prgEM.stEL3446_IO_1.MDP5001_342_Input.MDP5001_342_I1_Channel_Overcurrent					:=	MDP5001_342_I1_Channel_Overcurrent_1;
prgEM.stEL3446_IO_1.MDP5001_342_Input.MDP5001_342_I1_Channel_Inaccurate_Current			:=	MDP5001_342_I1_Channel_Inaccurate_Current_1;
prgEM.stEL3446_IO_1.MDP5001_342_Input.MDP5001_342_I1_Channel_Current_Guard_Warning		:=	MDP5001_342_I1_Channel_Current_Guard_Warning_1;
prgEM.stEL3446_IO_1.MDP5001_342_Input.MDP5001_342_I1_Channel_Current_Guard_Error			:=	MDP5001_342_I1_Channel_Current_Guard_Error_1;
prgEM.stEL3446_IO_1.MDP5001_342_Input.MDP5001_342_I1_Channel_Apparent_Power_Guard_Warning	:=	MDP5001_342_I1_Channel_Apparent_Power_Guard_Warning_1;
prgEM.stEL3446_IO_1.MDP5001_342_Input.MDP5001_342_I1_Channel_Apparent_Power_Guard_Error	:=	MDP5001_342_I1_Channel_Apparent_Power_Guard_Error_1;
prgEM.stEL3446_IO_1.MDP5001_342_Input.MDP5001_342_I1_Channel_Active_Power_Guard_Warning	:=	MDP5001_342_I1_Channel_Active_Power_Guard_Warning_1;
prgEM.stEL3446_IO_1.MDP5001_342_Input.MDP5001_342_I1_Channel_Active_Power_Guard_Error		:=	MDP5001_342_I1_Channel_Active_Power_Guard_Error_1;
prgEM.stEL3446_IO_1.MDP5001_342_Input.MDP5001_342_I1_Channel_Reactive_Power_Guard_Warning	:=	MDP5001_342_I1_Channel_Reactive_Power_Guard_Warning_1;
prgEM.stEL3446_IO_1.MDP5001_342_Input.MDP5001_342_I1_Channel_Reactive_Power_Guard_Error	:=	MDP5001_342_I1_Channel_Reactive_Power_Guard_Error_1;
prgEM.stEL3446_IO_1.MDP5001_342_Input.MDP5001_342_I1_Channel_DPM_Inaccurate				:=	MDP5001_342_I1_Channel_DPM_Inaccurate_1;
prgEM.stEL3446_IO_1.MDP5001_342_Input.MDP5001_342_I1_Channel_DPM_Timeout					:=	MDP5001_342_I1_Channel_DPM_Timeout_1;
prgEM.stEL3446_IO_1.MDP5001_342_Input.MDP5001_342_I1_Channel_TxPDO_Toggle					:=	MDP5001_342_I1_Channel_TxPDO_Toggle_1;
prgEM.stEL3446_IO_1.MDP5001_342_Input.MDP5001_342_I1_Channel_Current						:=	MDP5001_342_I1_Channel_Current_1;
prgEM.stEL3446_IO_1.MDP5001_342_Input.MDP5001_342_I1_Channel_Active_Power					:=	MDP5001_342_I1_Channel_Active_Power_1;
prgEM.stEL3446_IO_1.MDP5001_342_Input.MDP5001_342_I1_Channel_Apparent_Power				:=	MDP5001_342_I1_Channel_Apparent_Power_1;
prgEM.stEL3446_IO_1.MDP5001_342_Input.MDP5001_342_I1_Channel_Reactive_Power_Fundamental	:=	MDP5001_342_I1_Channel_Reactive_Power_Fundamental_1;
prgEM.stEL3446_IO_1.MDP5001_342_Input.MDP5001_342_I1_Channel_Active_Energy				:=	MDP5001_342_I1_Channel_Active_Energy_1;
prgEM.stEL3446_IO_1.MDP5001_342_Input.MDP5001_342_I2_Channel_Overcurrent					:=	MDP5001_342_I2_Channel_Overcurrent_1;
prgEM.stEL3446_IO_1.MDP5001_342_Input.MDP5001_342_I2_Channel_Inaccurate_Current			:=	MDP5001_342_I2_Channel_Inaccurate_Current_1;
prgEM.stEL3446_IO_1.MDP5001_342_Input.MDP5001_342_I2_Channel_Current_Guard_Warning		:=	MDP5001_342_I2_Channel_Current_Guard_Warning_1;
prgEM.stEL3446_IO_1.MDP5001_342_Input.MDP5001_342_I2_Channel_Current_Guard_Error			:=	MDP5001_342_I2_Channel_Current_Guard_Error_1;
prgEM.stEL3446_IO_1.MDP5001_342_Input.MDP5001_342_I2_Channel_Apparent_Power_Guard_Warning	:=	MDP5001_342_I2_Channel_Apparent_Power_Guard_Warning_1;
prgEM.stEL3446_IO_1.MDP5001_342_Input.MDP5001_342_I2_Channel_Apparent_Power_Guard_Error	:=	MDP5001_342_I2_Channel_Apparent_Power_Guard_Error_1;
prgEM.stEL3446_IO_1.MDP5001_342_Input.MDP5001_342_I2_Channel_Active_Power_Guard_Warning	:=	MDP5001_342_I2_Channel_Active_Power_Guard_Warning_1;
prgEM.stEL3446_IO_1.MDP5001_342_Input.MDP5001_342_I2_Channel_Active_Power_Guard_Error		:=	MDP5001_342_I2_Channel_Active_Power_Guard_Error_1;
prgEM.stEL3446_IO_1.MDP5001_342_Input.MDP5001_342_I2_Channel_Reactive_Power_Guard_Warning	:=	MDP5001_342_I2_Channel_Reactive_Power_Guard_Warning_1;
prgEM.stEL3446_IO_1.MDP5001_342_Input.MDP5001_342_I2_Channel_Reactive_Power_Guard_Error	:=	MDP5001_342_I2_Channel_Reactive_Power_Guard_Error_1;
prgEM.stEL3446_IO_1.MDP5001_342_Input.MDP5001_342_I2_Channel_DPM_Inaccurate				:=	MDP5001_342_I2_Channel_DPM_Inaccurate_1;
prgEM.stEL3446_IO_1.MDP5001_342_Input.MDP5001_342_I2_Channel_DPM_Timeout					:=	MDP5001_342_I2_Channel_DPM_Timeout_1;
prgEM.stEL3446_IO_1.MDP5001_342_Input.MDP5001_342_I2_Channel_TxPDO_Toggle					:=	MDP5001_342_I2_Channel_TxPDO_Toggle_1;
prgEM.stEL3446_IO_1.MDP5001_342_Input.MDP5001_342_I2_Channel_Current						:=	MDP5001_342_I2_Channel_Current_1;
prgEM.stEL3446_IO_1.MDP5001_342_Input.MDP5001_342_I2_Channel_Active_Power					:=	MDP5001_342_I2_Channel_Active_Power_1;
prgEM.stEL3446_IO_1.MDP5001_342_Input.MDP5001_342_I2_Channel_Apparent_Power				:=	MDP5001_342_I2_Channel_Apparent_Power_1;
prgEM.stEL3446_IO_1.MDP5001_342_Input.MDP5001_342_I2_Channel_Reactive_Power_Fundamental	:=	MDP5001_342_I2_Channel_Reactive_Power_Fundamental_1;
prgEM.stEL3446_IO_1.MDP5001_342_Input.MDP5001_342_I2_Channel_Active_Energy				:=	MDP5001_342_I2_Channel_Active_Energy_1;
prgEM.stEL3446_IO_1.MDP5001_342_Input.MDP5001_342_I3_Channel_Overcurrent					:=	MDP5001_342_I3_Channel_Overcurrent_1;
prgEM.stEL3446_IO_1.MDP5001_342_Input.MDP5001_342_I3_Channel_Inaccurate_Current			:=	MDP5001_342_I3_Channel_Inaccurate_Current_1;
prgEM.stEL3446_IO_1.MDP5001_342_Input.MDP5001_342_I3_Channel_Current_Guard_Warning		:=	MDP5001_342_I3_Channel_Current_Guard_Warning_1;
prgEM.stEL3446_IO_1.MDP5001_342_Input.MDP5001_342_I3_Channel_Current_Guard_Error			:=	MDP5001_342_I3_Channel_Current_Guard_Error_1;
prgEM.stEL3446_IO_1.MDP5001_342_Input.MDP5001_342_I3_Channel_Apparent_Power_Guard_Warning	:=	MDP5001_342_I3_Channel_Apparent_Power_Guard_Warning_1;
prgEM.stEL3446_IO_1.MDP5001_342_Input.MDP5001_342_I3_Channel_Apparent_Power_Guard_Error	:=	MDP5001_342_I3_Channel_Apparent_Power_Guard_Error_1;
prgEM.stEL3446_IO_1.MDP5001_342_Input.MDP5001_342_I3_Channel_Active_Power_Guard_Warning	:=	MDP5001_342_I3_Channel_Active_Power_Guard_Warning_1;
prgEM.stEL3446_IO_1.MDP5001_342_Input.MDP5001_342_I3_Channel_Active_Power_Guard_Error		:=	MDP5001_342_I3_Channel_Active_Power_Guard_Error_1;
prgEM.stEL3446_IO_1.MDP5001_342_Input.MDP5001_342_I3_Channel_Reactive_Power_Guard_Warning	:=	MDP5001_342_I3_Channel_Reactive_Power_Guard_Warning_1;
prgEM.stEL3446_IO_1.MDP5001_342_Input.MDP5001_342_I3_Channel_Reactive_Power_Guard_Error	:=	MDP5001_342_I3_Channel_Reactive_Power_Guard_Error_1;
prgEM.stEL3446_IO_1.MDP5001_342_Input.MDP5001_342_I3_Channel_DPM_Inaccurate				:=	MDP5001_342_I3_Channel_DPM_Inaccurate_1;
prgEM.stEL3446_IO_1.MDP5001_342_Input.MDP5001_342_I3_Channel_DPM_Timeout					:=	MDP5001_342_I3_Channel_DPM_Timeout_1;
prgEM.stEL3446_IO_1.MDP5001_342_Input.MDP5001_342_I3_Channel_TxPDO_Toggle					:=	MDP5001_342_I3_Channel_TxPDO_Toggle_1;
prgEM.stEL3446_IO_1.MDP5001_342_Input.MDP5001_342_I3_Channel_Current						:=	MDP5001_342_I3_Channel_Current_1;
prgEM.stEL3446_IO_1.MDP5001_342_Input.MDP5001_342_I3_Channel_Active_Power					:=	MDP5001_342_I3_Channel_Active_Power_1;
prgEM.stEL3446_IO_1.MDP5001_342_Input.MDP5001_342_I3_Channel_Apparent_Power				:=	MDP5001_342_I3_Channel_Apparent_Power_1;
prgEM.stEL3446_IO_1.MDP5001_342_Input.MDP5001_342_I3_Channel_Reactive_Power_Fundamental	:=	MDP5001_342_I3_Channel_Reactive_Power_Fundamental_1;
prgEM.stEL3446_IO_1.MDP5001_342_Input.MDP5001_342_I3_Channel_Active_Energy				:=	MDP5001_342_I3_Channel_Active_Energy_1;
prgEM.stEL3446_IO_1.MDP5001_342_Input.MDP5001_342_I4_Channel_Overcurrent					:=	MDP5001_342_I4_Channel_Overcurrent_1;
prgEM.stEL3446_IO_1.MDP5001_342_Input.MDP5001_342_I4_Channel_Inaccurate_Current			:=	MDP5001_342_I4_Channel_Inaccurate_Current_1;
prgEM.stEL3446_IO_1.MDP5001_342_Input.MDP5001_342_I4_Channel_Current_Guard_Warning		:=	MDP5001_342_I4_Channel_Current_Guard_Warning_1;
prgEM.stEL3446_IO_1.MDP5001_342_Input.MDP5001_342_I4_Channel_Current_Guard_Error			:=	MDP5001_342_I4_Channel_Current_Guard_Error_1;
prgEM.stEL3446_IO_1.MDP5001_342_Input.MDP5001_342_I4_Channel_Apparent_Power_Guard_Warning	:=	MDP5001_342_I4_Channel_Apparent_Power_Guard_Warning_1;
prgEM.stEL3446_IO_1.MDP5001_342_Input.MDP5001_342_I4_Channel_Apparent_Power_Guard_Error	:=	MDP5001_342_I4_Channel_Apparent_Power_Guard_Error_1;
prgEM.stEL3446_IO_1.MDP5001_342_Input.MDP5001_342_I4_Channel_Active_Power_Guard_Warning	:=	MDP5001_342_I4_Channel_Active_Power_Guard_Warning_1;
prgEM.stEL3446_IO_1.MDP5001_342_Input.MDP5001_342_I4_Channel_Active_Power_Guard_Error		:=	MDP5001_342_I4_Channel_Active_Power_Guard_Error_1;
prgEM.stEL3446_IO_1.MDP5001_342_Input.MDP5001_342_I4_Channel_Reactive_Power_Guard_Warning	:=	MDP5001_342_I4_Channel_Reactive_Power_Guard_Warning_1;
prgEM.stEL3446_IO_1.MDP5001_342_Input.MDP5001_342_I4_Channel_Reactive_Power_Guard_Error	:=	MDP5001_342_I4_Channel_Reactive_Power_Guard_Error_1;
prgEM.stEL3446_IO_1.MDP5001_342_Input.MDP5001_342_I4_Channel_DPM_Inaccurate				:=	MDP5001_342_I4_Channel_DPM_Inaccurate_1;
prgEM.stEL3446_IO_1.MDP5001_342_Input.MDP5001_342_I4_Channel_DPM_Timeout					:=	MDP5001_342_I4_Channel_DPM_Timeout_1;
prgEM.stEL3446_IO_1.MDP5001_342_Input.MDP5001_342_I4_Channel_TxPDO_Toggle					:=	MDP5001_342_I4_Channel_TxPDO_Toggle_1;
prgEM.stEL3446_IO_1.MDP5001_342_Input.MDP5001_342_I4_Channel_Current						:=	MDP5001_342_I4_Channel_Current_1;
prgEM.stEL3446_IO_1.MDP5001_342_Input.MDP5001_342_I4_Channel_Active_Power					:=	MDP5001_342_I4_Channel_Active_Power_1;
prgEM.stEL3446_IO_1.MDP5001_342_Input.MDP5001_342_I4_Channel_Apparent_Power				:=	MDP5001_342_I4_Channel_Apparent_Power_1;
prgEM.stEL3446_IO_1.MDP5001_342_Input.MDP5001_342_I4_Channel_Reactive_Power_Fundamental	:=	MDP5001_342_I4_Channel_Reactive_Power_Fundamental_1;
prgEM.stEL3446_IO_1.MDP5001_342_Input.MDP5001_342_I4_Channel_Active_Energy				:=	MDP5001_342_I4_Channel_Active_Energy_1;
prgEM.stEL3446_IO_1.MDP5001_342_Input.MDP5001_342_I5_Channel_Overcurrent					:=	MDP5001_342_I5_Channel_Overcurrent_1;
prgEM.stEL3446_IO_1.MDP5001_342_Input.MDP5001_342_I5_Channel_Inaccurate_Current			:=	MDP5001_342_I5_Channel_Inaccurate_Current_1;
prgEM.stEL3446_IO_1.MDP5001_342_Input.MDP5001_342_I5_Channel_Current_Guard_Warning		:=	MDP5001_342_I5_Channel_Current_Guard_Warning_1;
prgEM.stEL3446_IO_1.MDP5001_342_Input.MDP5001_342_I5_Channel_Current_Guard_Error			:=	MDP5001_342_I5_Channel_Current_Guard_Error_1;
prgEM.stEL3446_IO_1.MDP5001_342_Input.MDP5001_342_I5_Channel_Apparent_Power_Guard_Warning	:=	MDP5001_342_I5_Channel_Apparent_Power_Guard_Warning_1;
prgEM.stEL3446_IO_1.MDP5001_342_Input.MDP5001_342_I5_Channel_Apparent_Power_Guard_Error	:=	MDP5001_342_I5_Channel_Apparent_Power_Guard_Error_1;
prgEM.stEL3446_IO_1.MDP5001_342_Input.MDP5001_342_I5_Channel_Active_Power_Guard_Warning	:=	MDP5001_342_I5_Channel_Active_Power_Guard_Warning_1;
prgEM.stEL3446_IO_1.MDP5001_342_Input.MDP5001_342_I5_Channel_Active_Power_Guard_Error		:=	MDP5001_342_I5_Channel_Active_Power_Guard_Error_1;
prgEM.stEL3446_IO_1.MDP5001_342_Input.MDP5001_342_I5_Channel_Reactive_Power_Guard_Warning	:=	MDP5001_342_I5_Channel_Reactive_Power_Guard_Warning_1;
prgEM.stEL3446_IO_1.MDP5001_342_Input.MDP5001_342_I5_Channel_Reactive_Power_Guard_Error	:=	MDP5001_342_I5_Channel_Reactive_Power_Guard_Error_1;
prgEM.stEL3446_IO_1.MDP5001_342_Input.MDP5001_342_I5_Channel_DPM_Inaccurate				:=	MDP5001_342_I5_Channel_DPM_Inaccurate_1;
prgEM.stEL3446_IO_1.MDP5001_342_Input.MDP5001_342_I5_Channel_DPM_Timeout					:=	MDP5001_342_I5_Channel_DPM_Timeout_1;
prgEM.stEL3446_IO_1.MDP5001_342_Input.MDP5001_342_I5_Channel_TxPDO_Toggle					:=	MDP5001_342_I5_Channel_TxPDO_Toggle_1;
prgEM.stEL3446_IO_1.MDP5001_342_Input.MDP5001_342_I5_Channel_Current						:=	MDP5001_342_I5_Channel_Current_1;
prgEM.stEL3446_IO_1.MDP5001_342_Input.MDP5001_342_I5_Channel_Active_Power					:=	MDP5001_342_I5_Channel_Active_Power_1;
prgEM.stEL3446_IO_1.MDP5001_342_Input.MDP5001_342_I5_Channel_Apparent_Power				:=	MDP5001_342_I5_Channel_Apparent_Power_1;
prgEM.stEL3446_IO_1.MDP5001_342_Input.MDP5001_342_I5_Channel_Reactive_Power_Fundamental	:=	MDP5001_342_I5_Channel_Reactive_Power_Fundamental_1;
prgEM.stEL3446_IO_1.MDP5001_342_Input.MDP5001_342_I5_Channel_Active_Energy				:=	MDP5001_342_I5_Channel_Active_Energy_1;
prgEM.stEL3446_IO_1.MDP5001_342_Input.MDP5001_342_I6_Channel_Overcurrent					:=	MDP5001_342_I6_Channel_Overcurrent_1;
prgEM.stEL3446_IO_1.MDP5001_342_Input.MDP5001_342_I6_Channel_Inaccurate_Current			:=	MDP5001_342_I6_Channel_Inaccurate_Current_1;
prgEM.stEL3446_IO_1.MDP5001_342_Input.MDP5001_342_I6_Channel_Current_Guard_Warning		:=	MDP5001_342_I6_Channel_Current_Guard_Warning_1;
prgEM.stEL3446_IO_1.MDP5001_342_Input.MDP5001_342_I6_Channel_Current_Guard_Error			:=	MDP5001_342_I6_Channel_Current_Guard_Error_1;
prgEM.stEL3446_IO_1.MDP5001_342_Input.MDP5001_342_I6_Channel_Apparent_Power_Guard_Warning	:=	MDP5001_342_I6_Channel_Apparent_Power_Guard_Warning_1;
prgEM.stEL3446_IO_1.MDP5001_342_Input.MDP5001_342_I6_Channel_Apparent_Power_Guard_Error	:=	MDP5001_342_I6_Channel_Apparent_Power_Guard_Error_1;
prgEM.stEL3446_IO_1.MDP5001_342_Input.MDP5001_342_I6_Channel_Active_Power_Guard_Warning	:=	MDP5001_342_I6_Channel_Active_Power_Guard_Warning_1;
prgEM.stEL3446_IO_1.MDP5001_342_Input.MDP5001_342_I6_Channel_Active_Power_Guard_Error		:=	MDP5001_342_I6_Channel_Active_Power_Guard_Error_1;
prgEM.stEL3446_IO_1.MDP5001_342_Input.MDP5001_342_I6_Channel_Reactive_Power_Guard_Warning	:=	MDP5001_342_I6_Channel_Reactive_Power_Guard_Warning_1;
prgEM.stEL3446_IO_1.MDP5001_342_Input.MDP5001_342_I6_Channel_Reactive_Power_Guard_Error	:=	MDP5001_342_I6_Channel_Reactive_Power_Guard_Error_1;
prgEM.stEL3446_IO_1.MDP5001_342_Input.MDP5001_342_I6_Channel_DPM_Inaccurate				:=	MDP5001_342_I6_Channel_DPM_Inaccurate_1;
prgEM.stEL3446_IO_1.MDP5001_342_Input.MDP5001_342_I6_Channel_DPM_Timeout					:=	MDP5001_342_I6_Channel_DPM_Timeout_1;
prgEM.stEL3446_IO_1.MDP5001_342_Input.MDP5001_342_I6_Channel_TxPDO_Toggle					:=	MDP5001_342_I6_Channel_TxPDO_Toggle_1;
prgEM.stEL3446_IO_1.MDP5001_342_Input.MDP5001_342_I6_Channel_Current						:=	MDP5001_342_I6_Channel_Current_1;
prgEM.stEL3446_IO_1.MDP5001_342_Input.MDP5001_342_I6_Channel_Active_Power					:=	MDP5001_342_I6_Channel_Active_Power_1;
prgEM.stEL3446_IO_1.MDP5001_342_Input.MDP5001_342_I6_Channel_Apparent_Power				:=	MDP5001_342_I6_Channel_Apparent_Power_1;
prgEM.stEL3446_IO_1.MDP5001_342_Input.MDP5001_342_I6_Channel_Reactive_Power_Fundamental	:=	MDP5001_342_I6_Channel_Reactive_Power_Fundamental_1;
prgEM.stEL3446_IO_1.MDP5001_342_Input.MDP5001_342_I6_Channel_Active_Energy				:=	MDP5001_342_I6_Channel_Active_Energy_1;
prgEM.stEL3446_IO_1.MDP5001_342_Input.MDP5001_342_DPM_Variant_Value_In_TxPDO_Toggle		:=	MDP5001_342_DPM_Variant_Value_In_TxPDO_Toggle_1;
prgEM.stEL3446_IO_1.MDP5001_342_Input.MDP5001_342_DPM_Variant_Value_In_Index_1_REAL		:=	MDP5001_342_DPM_Variant_Value_In_Index_1_REAL_1;
prgEM.stEL3446_IO_1.MDP5001_342_Input.MDP5001_342_DPM_Variant_Value_In_Value_1_REAL		:=	MDP5001_342_DPM_Variant_Value_In_Value_1_REAL_1;
prgEM.stEL3446_IO_1.MDP5001_342_Input.MDP5001_342_DPM_Variant_Value_In_Index_2_REAL		:=	MDP5001_342_DPM_Variant_Value_In_Index_2_REAL_1;
prgEM.stEL3446_IO_1.MDP5001_342_Input.MDP5001_342_DPM_Variant_Value_In_Value_2_REAL		:=	MDP5001_342_DPM_Variant_Value_In_Value_2_REAL_1;
prgEM.stEL3446_IO_1.MDP5001_342_Input.MDP5001_342_DPM_Variant_Value_In_Index_3_REAL		:=	MDP5001_342_DPM_Variant_Value_In_Index_3_REAL_1;
prgEM.stEL3446_IO_1.MDP5001_342_Input.MDP5001_342_DPM_Variant_Value_In_Value_3_REAL		:=	MDP5001_342_DPM_Variant_Value_In_Value_3_REAL_1;
prgEM.stEL3446_IO_1.MDP5001_342_Input.MDP5001_342_DPM_Variant_Value_In_Index_4_ULINT		:=	MDP5001_342_DPM_Variant_Value_In_Index_4_ULINT_1;
prgEM.stEL3446_IO_1.MDP5001_342_Input.MDP5001_342_DPM_Variant_Value_In_Value_4_ULINT		:=	MDP5001_342_DPM_Variant_Value_In_Value_4_ULINT_1;

MDP5001_342_DPM_Variant_Value_Out_Index_1_REAL_1	:= 		prgEM.stEL3446_IO_1.MDP5001_342_Output.MDP5001_342_DPM_Variant_Value_Out_Index_1_REAL	;
MDP5001_342_DPM_Variant_Value_Out_Index_2_REAL_1	:= 		prgEM.stEL3446_IO_1.MDP5001_342_Output.MDP5001_342_DPM_Variant_Value_Out_Index_2_REAL	;	
MDP5001_342_DPM_Variant_Value_Out_Index_3_REAL_1	:= 		prgEM.stEL3446_IO_1.MDP5001_342_Output.MDP5001_342_DPM_Variant_Value_Out_Index_3_REAL	;
MDP5001_342_DPM_Variant_Value_Out_Index_4_ULINT_1	:= 		prgEM.stEL3446_IO_1.MDP5001_342_Output.MDP5001_342_DPM_Variant_Value_Out_Index_4_ULINT	;
MDP5001_342_DPM_Data_Data_1_1						:= 		prgEM.stEL3446_IO_1.MDP5001_342_Output.MDP5001_342_DPM_Data_Data_1	;
MDP5001_342_DPM_Data_Data_2_1						:= 		prgEM.stEL3446_IO_1.MDP5001_342_Output.MDP5001_342_DPM_Data_Data_2	;
MDP5001_342_DPM_Data_Data_3_1						:= 		prgEM.stEL3446_IO_1.MDP5001_342_Output.MDP5001_342_DPM_Data_Data_3	;
MDP5001_342_DPM_Data_Data_4_1						:= 		prgEM.stEL3446_IO_1.MDP5001_342_Output.MDP5001_342_DPM_Data_Data_4	;
MDP5001_342_DPM_Data_Data_5_1						:= 		prgEM.stEL3446_IO_1.MDP5001_342_Output.MDP5001_342_DPM_Data_Data_5	;
MDP5001_342_DPM_Data_Data_6_1						:= 		prgEM.stEL3446_IO_1.MDP5001_342_Output.MDP5001_342_DPM_Data_Data_6	;
MDP5001_342_DPM_Data_Data_7_1						:= 		prgEM.stEL3446_IO_1.MDP5001_342_Output.MDP5001_342_DPM_Data_Data_7	;
MDP5001_342_DPM_Data_Data_8_1						:= 		prgEM.stEL3446_IO_1.MDP5001_342_Output.MDP5001_342_DPM_Data_Data_8	;
MDP5001_342_DPM_Data_Data_9_1						:= 		prgEM.stEL3446_IO_1.MDP5001_342_Output.MDP5001_342_DPM_Data_Data_9	;
MDP5001_342_DPM_Data_Data_10_1						:= 		prgEM.stEL3446_IO_1.MDP5001_342_Output.MDP5001_342_DPM_Data_Data_10	;
MDP5001_342_DPM_Data_Data_11_1						:= 		prgEM.stEL3446_IO_1.MDP5001_342_Output.MDP5001_342_DPM_Data_Data_11	;
MDP5001_342_DPM_Data_Data_12_1						:= 		prgEM.stEL3446_IO_1.MDP5001_342_Output.MDP5001_342_DPM_Data_Data_12	;
MDP5001_342_DPM_Data_Data_13_1						:= 		prgEM.stEL3446_IO_1.MDP5001_342_Output.MDP5001_342_DPM_Data_Data_13	;
MDP5001_342_DPM_Data_Data_14_1						:= 		prgEM.stEL3446_IO_1.MDP5001_342_Output.MDP5001_342_DPM_Data_Data_14	;
MDP5001_342_DPM_Data_Data_15_1						:= 		prgEM.stEL3446_IO_1.MDP5001_342_Output.MDP5001_342_DPM_Data_Data_15	;
MDP5001_342_DPM_Data_Data_16_1						:= 		prgEM.stEL3446_IO_1.MDP5001_342_Output.MDP5001_342_DPM_Data_Data_16	;
MDP5001_342_DPM_Data_Data_17_1						:= 		prgEM.stEL3446_IO_1.MDP5001_342_Output.MDP5001_342_DPM_Data_Data_17	;
MDP5001_342_DPM_Data_Data_18_1						:= 		prgEM.stEL3446_IO_1.MDP5001_342_Output.MDP5001_342_DPM_Data_Data_18	;
MDP5001_342_DPM_Data_Data_19_1						:= 		prgEM.stEL3446_IO_1.MDP5001_342_Output.MDP5001_342_DPM_Data_Data_19	;
MDP5001_342_DPM_Data_Data_20_1						:= 		prgEM.stEL3446_IO_1.MDP5001_342_Output.MDP5001_342_DPM_Data_Data_20	;




prgEM.stEL3446_IO_2.MDP5001_342_Input.MDP5001_342_I1_Channel_Overcurrent					:=	MDP5001_342_I1_Channel_Overcurrent_2;
prgEM.stEL3446_IO_2.MDP5001_342_Input.MDP5001_342_I1_Channel_Inaccurate_Current			:=	MDP5001_342_I1_Channel_Inaccurate_Current_2;
prgEM.stEL3446_IO_2.MDP5001_342_Input.MDP5001_342_I1_Channel_Current_Guard_Warning		:=	MDP5001_342_I1_Channel_Current_Guard_Warning_2;
prgEM.stEL3446_IO_2.MDP5001_342_Input.MDP5001_342_I1_Channel_Current_Guard_Error			:=	MDP5001_342_I1_Channel_Current_Guard_Error_2;
prgEM.stEL3446_IO_2.MDP5001_342_Input.MDP5001_342_I1_Channel_Apparent_Power_Guard_Warning	:=	MDP5001_342_I1_Channel_Apparent_Power_Guard_Warning_2;
prgEM.stEL3446_IO_2.MDP5001_342_Input.MDP5001_342_I1_Channel_Apparent_Power_Guard_Error	:=	MDP5001_342_I1_Channel_Apparent_Power_Guard_Error_2;
prgEM.stEL3446_IO_2.MDP5001_342_Input.MDP5001_342_I1_Channel_Active_Power_Guard_Warning	:=	MDP5001_342_I1_Channel_Active_Power_Guard_Warning_2;
prgEM.stEL3446_IO_2.MDP5001_342_Input.MDP5001_342_I1_Channel_Active_Power_Guard_Error		:=	MDP5001_342_I1_Channel_Active_Power_Guard_Error_2;
prgEM.stEL3446_IO_2.MDP5001_342_Input.MDP5001_342_I1_Channel_Reactive_Power_Guard_Warning	:=	MDP5001_342_I1_Channel_Reactive_Power_Guard_Warning_2;
prgEM.stEL3446_IO_2.MDP5001_342_Input.MDP5001_342_I1_Channel_Reactive_Power_Guard_Error	:=	MDP5001_342_I1_Channel_Reactive_Power_Guard_Error_2;
prgEM.stEL3446_IO_2.MDP5001_342_Input.MDP5001_342_I1_Channel_DPM_Inaccurate				:=	MDP5001_342_I1_Channel_DPM_Inaccurate_2;
prgEM.stEL3446_IO_2.MDP5001_342_Input.MDP5001_342_I1_Channel_DPM_Timeout					:=	MDP5001_342_I1_Channel_DPM_Timeout_2;
prgEM.stEL3446_IO_2.MDP5001_342_Input.MDP5001_342_I1_Channel_TxPDO_Toggle					:=	MDP5001_342_I1_Channel_TxPDO_Toggle_2;
prgEM.stEL3446_IO_2.MDP5001_342_Input.MDP5001_342_I1_Channel_Current						:=	MDP5001_342_I1_Channel_Current_2;
prgEM.stEL3446_IO_2.MDP5001_342_Input.MDP5001_342_I1_Channel_Active_Power					:=	MDP5001_342_I1_Channel_Active_Power_2;
prgEM.stEL3446_IO_2.MDP5001_342_Input.MDP5001_342_I1_Channel_Apparent_Power				:=	MDP5001_342_I1_Channel_Apparent_Power_2;
prgEM.stEL3446_IO_2.MDP5001_342_Input.MDP5001_342_I1_Channel_Reactive_Power_Fundamental	:=	MDP5001_342_I1_Channel_Reactive_Power_Fundamental_2;
prgEM.stEL3446_IO_2.MDP5001_342_Input.MDP5001_342_I1_Channel_Active_Energy				:=	MDP5001_342_I1_Channel_Active_Energy_2;
prgEM.stEL3446_IO_2.MDP5001_342_Input.MDP5001_342_I2_Channel_Overcurrent					:=	MDP5001_342_I2_Channel_Overcurrent_2;
prgEM.stEL3446_IO_2.MDP5001_342_Input.MDP5001_342_I2_Channel_Inaccurate_Current			:=	MDP5001_342_I2_Channel_Inaccurate_Current_2;
prgEM.stEL3446_IO_2.MDP5001_342_Input.MDP5001_342_I2_Channel_Current_Guard_Warning		:=	MDP5001_342_I2_Channel_Current_Guard_Warning_2;
prgEM.stEL3446_IO_2.MDP5001_342_Input.MDP5001_342_I2_Channel_Current_Guard_Error			:=	MDP5001_342_I2_Channel_Current_Guard_Error_2;
prgEM.stEL3446_IO_2.MDP5001_342_Input.MDP5001_342_I2_Channel_Apparent_Power_Guard_Warning	:=	MDP5001_342_I2_Channel_Apparent_Power_Guard_Warning_2;
prgEM.stEL3446_IO_2.MDP5001_342_Input.MDP5001_342_I2_Channel_Apparent_Power_Guard_Error	:=	MDP5001_342_I2_Channel_Apparent_Power_Guard_Error_2;
prgEM.stEL3446_IO_2.MDP5001_342_Input.MDP5001_342_I2_Channel_Active_Power_Guard_Warning	:=	MDP5001_342_I2_Channel_Active_Power_Guard_Warning_2;
prgEM.stEL3446_IO_2.MDP5001_342_Input.MDP5001_342_I2_Channel_Active_Power_Guard_Error		:=	MDP5001_342_I2_Channel_Active_Power_Guard_Error_2;
prgEM.stEL3446_IO_2.MDP5001_342_Input.MDP5001_342_I2_Channel_Reactive_Power_Guard_Warning	:=	MDP5001_342_I2_Channel_Reactive_Power_Guard_Warning_2;
prgEM.stEL3446_IO_2.MDP5001_342_Input.MDP5001_342_I2_Channel_Reactive_Power_Guard_Error	:=	MDP5001_342_I2_Channel_Reactive_Power_Guard_Error_2;
prgEM.stEL3446_IO_2.MDP5001_342_Input.MDP5001_342_I2_Channel_DPM_Inaccurate				:=	MDP5001_342_I2_Channel_DPM_Inaccurate_2;
prgEM.stEL3446_IO_2.MDP5001_342_Input.MDP5001_342_I2_Channel_DPM_Timeout					:=	MDP5001_342_I2_Channel_DPM_Timeout_2;
prgEM.stEL3446_IO_2.MDP5001_342_Input.MDP5001_342_I2_Channel_TxPDO_Toggle					:=	MDP5001_342_I2_Channel_TxPDO_Toggle_2;
prgEM.stEL3446_IO_2.MDP5001_342_Input.MDP5001_342_I2_Channel_Current						:=	MDP5001_342_I2_Channel_Current_2;
prgEM.stEL3446_IO_2.MDP5001_342_Input.MDP5001_342_I2_Channel_Active_Power					:=	MDP5001_342_I2_Channel_Active_Power_2;
prgEM.stEL3446_IO_2.MDP5001_342_Input.MDP5001_342_I2_Channel_Apparent_Power				:=	MDP5001_342_I2_Channel_Apparent_Power_2;
prgEM.stEL3446_IO_2.MDP5001_342_Input.MDP5001_342_I2_Channel_Reactive_Power_Fundamental	:=	MDP5001_342_I2_Channel_Reactive_Power_Fundamental_2;
prgEM.stEL3446_IO_2.MDP5001_342_Input.MDP5001_342_I2_Channel_Active_Energy				:=	MDP5001_342_I2_Channel_Active_Energy_2;
prgEM.stEL3446_IO_2.MDP5001_342_Input.MDP5001_342_I3_Channel_Overcurrent					:=	MDP5001_342_I3_Channel_Overcurrent_2;
prgEM.stEL3446_IO_2.MDP5001_342_Input.MDP5001_342_I3_Channel_Inaccurate_Current			:=	MDP5001_342_I3_Channel_Inaccurate_Current_2;
prgEM.stEL3446_IO_2.MDP5001_342_Input.MDP5001_342_I3_Channel_Current_Guard_Warning		:=	MDP5001_342_I3_Channel_Current_Guard_Warning_2;
prgEM.stEL3446_IO_2.MDP5001_342_Input.MDP5001_342_I3_Channel_Current_Guard_Error			:=	MDP5001_342_I3_Channel_Current_Guard_Error_2;
prgEM.stEL3446_IO_2.MDP5001_342_Input.MDP5001_342_I3_Channel_Apparent_Power_Guard_Warning	:=	MDP5001_342_I3_Channel_Apparent_Power_Guard_Warning_2;
prgEM.stEL3446_IO_2.MDP5001_342_Input.MDP5001_342_I3_Channel_Apparent_Power_Guard_Error	:=	MDP5001_342_I3_Channel_Apparent_Power_Guard_Error_2;
prgEM.stEL3446_IO_2.MDP5001_342_Input.MDP5001_342_I3_Channel_Active_Power_Guard_Warning	:=	MDP5001_342_I3_Channel_Active_Power_Guard_Warning_2;
prgEM.stEL3446_IO_2.MDP5001_342_Input.MDP5001_342_I3_Channel_Active_Power_Guard_Error		:=	MDP5001_342_I3_Channel_Active_Power_Guard_Error_2;
prgEM.stEL3446_IO_2.MDP5001_342_Input.MDP5001_342_I3_Channel_Reactive_Power_Guard_Warning	:=	MDP5001_342_I3_Channel_Reactive_Power_Guard_Warning_2;
prgEM.stEL3446_IO_2.MDP5001_342_Input.MDP5001_342_I3_Channel_Reactive_Power_Guard_Error	:=	MDP5001_342_I3_Channel_Reactive_Power_Guard_Error_2;
prgEM.stEL3446_IO_2.MDP5001_342_Input.MDP5001_342_I3_Channel_DPM_Inaccurate				:=	MDP5001_342_I3_Channel_DPM_Inaccurate_2;
prgEM.stEL3446_IO_2.MDP5001_342_Input.MDP5001_342_I3_Channel_DPM_Timeout					:=	MDP5001_342_I3_Channel_DPM_Timeout_2;
prgEM.stEL3446_IO_2.MDP5001_342_Input.MDP5001_342_I3_Channel_TxPDO_Toggle					:=	MDP5001_342_I3_Channel_TxPDO_Toggle_2;
prgEM.stEL3446_IO_2.MDP5001_342_Input.MDP5001_342_I3_Channel_Current						:=	MDP5001_342_I3_Channel_Current_2;
prgEM.stEL3446_IO_2.MDP5001_342_Input.MDP5001_342_I3_Channel_Active_Power					:=	MDP5001_342_I3_Channel_Active_Power_2;
prgEM.stEL3446_IO_2.MDP5001_342_Input.MDP5001_342_I3_Channel_Apparent_Power				:=	MDP5001_342_I3_Channel_Apparent_Power_2;
prgEM.stEL3446_IO_2.MDP5001_342_Input.MDP5001_342_I3_Channel_Reactive_Power_Fundamental	:=	MDP5001_342_I3_Channel_Reactive_Power_Fundamental_2;
prgEM.stEL3446_IO_2.MDP5001_342_Input.MDP5001_342_I3_Channel_Active_Energy				:=	MDP5001_342_I3_Channel_Active_Energy_2;
prgEM.stEL3446_IO_2.MDP5001_342_Input.MDP5001_342_I4_Channel_Overcurrent					:=	MDP5001_342_I4_Channel_Overcurrent_2;
prgEM.stEL3446_IO_2.MDP5001_342_Input.MDP5001_342_I4_Channel_Inaccurate_Current			:=	MDP5001_342_I4_Channel_Inaccurate_Current_2;
prgEM.stEL3446_IO_2.MDP5001_342_Input.MDP5001_342_I4_Channel_Current_Guard_Warning		:=	MDP5001_342_I4_Channel_Current_Guard_Warning_2;
prgEM.stEL3446_IO_2.MDP5001_342_Input.MDP5001_342_I4_Channel_Current_Guard_Error			:=	MDP5001_342_I4_Channel_Current_Guard_Error_2;
prgEM.stEL3446_IO_2.MDP5001_342_Input.MDP5001_342_I4_Channel_Apparent_Power_Guard_Warning	:=	MDP5001_342_I4_Channel_Apparent_Power_Guard_Warning_2;
prgEM.stEL3446_IO_2.MDP5001_342_Input.MDP5001_342_I4_Channel_Apparent_Power_Guard_Error	:=	MDP5001_342_I4_Channel_Apparent_Power_Guard_Error_2;
prgEM.stEL3446_IO_2.MDP5001_342_Input.MDP5001_342_I4_Channel_Active_Power_Guard_Warning	:=	MDP5001_342_I4_Channel_Active_Power_Guard_Warning_2;
prgEM.stEL3446_IO_2.MDP5001_342_Input.MDP5001_342_I4_Channel_Active_Power_Guard_Error		:=	MDP5001_342_I4_Channel_Active_Power_Guard_Error_2;
prgEM.stEL3446_IO_2.MDP5001_342_Input.MDP5001_342_I4_Channel_Reactive_Power_Guard_Warning	:=	MDP5001_342_I4_Channel_Reactive_Power_Guard_Warning_2;
prgEM.stEL3446_IO_2.MDP5001_342_Input.MDP5001_342_I4_Channel_Reactive_Power_Guard_Error	:=	MDP5001_342_I4_Channel_Reactive_Power_Guard_Error_2;
prgEM.stEL3446_IO_2.MDP5001_342_Input.MDP5001_342_I4_Channel_DPM_Inaccurate				:=	MDP5001_342_I4_Channel_DPM_Inaccurate_2;
prgEM.stEL3446_IO_2.MDP5001_342_Input.MDP5001_342_I4_Channel_DPM_Timeout					:=	MDP5001_342_I4_Channel_DPM_Timeout_2;
prgEM.stEL3446_IO_2.MDP5001_342_Input.MDP5001_342_I4_Channel_TxPDO_Toggle					:=	MDP5001_342_I4_Channel_TxPDO_Toggle_2;
prgEM.stEL3446_IO_2.MDP5001_342_Input.MDP5001_342_I4_Channel_Current						:=	MDP5001_342_I4_Channel_Current_2;
prgEM.stEL3446_IO_2.MDP5001_342_Input.MDP5001_342_I4_Channel_Active_Power					:=	MDP5001_342_I4_Channel_Active_Power_2;
prgEM.stEL3446_IO_2.MDP5001_342_Input.MDP5001_342_I4_Channel_Apparent_Power				:=	MDP5001_342_I4_Channel_Apparent_Power_2;
prgEM.stEL3446_IO_2.MDP5001_342_Input.MDP5001_342_I4_Channel_Reactive_Power_Fundamental	:=	MDP5001_342_I4_Channel_Reactive_Power_Fundamental_2;
prgEM.stEL3446_IO_2.MDP5001_342_Input.MDP5001_342_I4_Channel_Active_Energy				:=	MDP5001_342_I4_Channel_Active_Energy_2;
prgEM.stEL3446_IO_2.MDP5001_342_Input.MDP5001_342_I5_Channel_Overcurrent					:=	MDP5001_342_I5_Channel_Overcurrent_2;
prgEM.stEL3446_IO_2.MDP5001_342_Input.MDP5001_342_I5_Channel_Inaccurate_Current			:=	MDP5001_342_I5_Channel_Inaccurate_Current_2;
prgEM.stEL3446_IO_2.MDP5001_342_Input.MDP5001_342_I5_Channel_Current_Guard_Warning		:=	MDP5001_342_I5_Channel_Current_Guard_Warning_2;
prgEM.stEL3446_IO_2.MDP5001_342_Input.MDP5001_342_I5_Channel_Current_Guard_Error			:=	MDP5001_342_I5_Channel_Current_Guard_Error_2;
prgEM.stEL3446_IO_2.MDP5001_342_Input.MDP5001_342_I5_Channel_Apparent_Power_Guard_Warning	:=	MDP5001_342_I5_Channel_Apparent_Power_Guard_Warning_2;
prgEM.stEL3446_IO_2.MDP5001_342_Input.MDP5001_342_I5_Channel_Apparent_Power_Guard_Error	:=	MDP5001_342_I5_Channel_Apparent_Power_Guard_Error_2;
prgEM.stEL3446_IO_2.MDP5001_342_Input.MDP5001_342_I5_Channel_Active_Power_Guard_Warning	:=	MDP5001_342_I5_Channel_Active_Power_Guard_Warning_2;
prgEM.stEL3446_IO_2.MDP5001_342_Input.MDP5001_342_I5_Channel_Active_Power_Guard_Error		:=	MDP5001_342_I5_Channel_Active_Power_Guard_Error_2;
prgEM.stEL3446_IO_2.MDP5001_342_Input.MDP5001_342_I5_Channel_Reactive_Power_Guard_Warning	:=	MDP5001_342_I5_Channel_Reactive_Power_Guard_Warning_2;
prgEM.stEL3446_IO_2.MDP5001_342_Input.MDP5001_342_I5_Channel_Reactive_Power_Guard_Error	:=	MDP5001_342_I5_Channel_Reactive_Power_Guard_Error_2;
prgEM.stEL3446_IO_2.MDP5001_342_Input.MDP5001_342_I5_Channel_DPM_Inaccurate				:=	MDP5001_342_I5_Channel_DPM_Inaccurate_2;
prgEM.stEL3446_IO_2.MDP5001_342_Input.MDP5001_342_I5_Channel_DPM_Timeout					:=	MDP5001_342_I5_Channel_DPM_Timeout_2;
prgEM.stEL3446_IO_2.MDP5001_342_Input.MDP5001_342_I5_Channel_TxPDO_Toggle					:=	MDP5001_342_I5_Channel_TxPDO_Toggle_2;
prgEM.stEL3446_IO_2.MDP5001_342_Input.MDP5001_342_I5_Channel_Current						:=	MDP5001_342_I5_Channel_Current_2;
prgEM.stEL3446_IO_2.MDP5001_342_Input.MDP5001_342_I5_Channel_Active_Power					:=	MDP5001_342_I5_Channel_Active_Power_2;
prgEM.stEL3446_IO_2.MDP5001_342_Input.MDP5001_342_I5_Channel_Apparent_Power				:=	MDP5001_342_I5_Channel_Apparent_Power_2;
prgEM.stEL3446_IO_2.MDP5001_342_Input.MDP5001_342_I5_Channel_Reactive_Power_Fundamental	:=	MDP5001_342_I5_Channel_Reactive_Power_Fundamental_2;
prgEM.stEL3446_IO_2.MDP5001_342_Input.MDP5001_342_I5_Channel_Active_Energy				:=	MDP5001_342_I5_Channel_Active_Energy_2;
prgEM.stEL3446_IO_2.MDP5001_342_Input.MDP5001_342_I6_Channel_Overcurrent					:=	MDP5001_342_I6_Channel_Overcurrent_2;
prgEM.stEL3446_IO_2.MDP5001_342_Input.MDP5001_342_I6_Channel_Inaccurate_Current			:=	MDP5001_342_I6_Channel_Inaccurate_Current_2;
prgEM.stEL3446_IO_2.MDP5001_342_Input.MDP5001_342_I6_Channel_Current_Guard_Warning		:=	MDP5001_342_I6_Channel_Current_Guard_Warning_2;
prgEM.stEL3446_IO_2.MDP5001_342_Input.MDP5001_342_I6_Channel_Current_Guard_Error			:=	MDP5001_342_I6_Channel_Current_Guard_Error_2;
prgEM.stEL3446_IO_2.MDP5001_342_Input.MDP5001_342_I6_Channel_Apparent_Power_Guard_Warning	:=	MDP5001_342_I6_Channel_Apparent_Power_Guard_Warning_2;
prgEM.stEL3446_IO_2.MDP5001_342_Input.MDP5001_342_I6_Channel_Apparent_Power_Guard_Error	:=	MDP5001_342_I6_Channel_Apparent_Power_Guard_Error_2;
prgEM.stEL3446_IO_2.MDP5001_342_Input.MDP5001_342_I6_Channel_Active_Power_Guard_Warning	:=	MDP5001_342_I6_Channel_Active_Power_Guard_Warning_2;
prgEM.stEL3446_IO_2.MDP5001_342_Input.MDP5001_342_I6_Channel_Active_Power_Guard_Error		:=	MDP5001_342_I6_Channel_Active_Power_Guard_Error_2;
prgEM.stEL3446_IO_2.MDP5001_342_Input.MDP5001_342_I6_Channel_Reactive_Power_Guard_Warning	:=	MDP5001_342_I6_Channel_Reactive_Power_Guard_Warning_2;
prgEM.stEL3446_IO_2.MDP5001_342_Input.MDP5001_342_I6_Channel_Reactive_Power_Guard_Error	:=	MDP5001_342_I6_Channel_Reactive_Power_Guard_Error_2;
prgEM.stEL3446_IO_2.MDP5001_342_Input.MDP5001_342_I6_Channel_DPM_Inaccurate				:=	MDP5001_342_I6_Channel_DPM_Inaccurate_2;
prgEM.stEL3446_IO_2.MDP5001_342_Input.MDP5001_342_I6_Channel_DPM_Timeout					:=	MDP5001_342_I6_Channel_DPM_Timeout_2;
prgEM.stEL3446_IO_2.MDP5001_342_Input.MDP5001_342_I6_Channel_TxPDO_Toggle					:=	MDP5001_342_I6_Channel_TxPDO_Toggle_2;
prgEM.stEL3446_IO_2.MDP5001_342_Input.MDP5001_342_I6_Channel_Current						:=	MDP5001_342_I6_Channel_Current_2;
prgEM.stEL3446_IO_2.MDP5001_342_Input.MDP5001_342_I6_Channel_Active_Power					:=	MDP5001_342_I6_Channel_Active_Power_2;
prgEM.stEL3446_IO_2.MDP5001_342_Input.MDP5001_342_I6_Channel_Apparent_Power				:=	MDP5001_342_I6_Channel_Apparent_Power_2;
prgEM.stEL3446_IO_2.MDP5001_342_Input.MDP5001_342_I6_Channel_Reactive_Power_Fundamental	:=	MDP5001_342_I6_Channel_Reactive_Power_Fundamental_2;
prgEM.stEL3446_IO_2.MDP5001_342_Input.MDP5001_342_I6_Channel_Active_Energy				:=	MDP5001_342_I6_Channel_Active_Energy_2;
prgEM.stEL3446_IO_2.MDP5001_342_Input.MDP5001_342_DPM_Variant_Value_In_TxPDO_Toggle		:=	MDP5001_342_DPM_Variant_Value_In_TxPDO_Toggle_2;
prgEM.stEL3446_IO_2.MDP5001_342_Input.MDP5001_342_DPM_Variant_Value_In_Index_1_REAL		:=	MDP5001_342_DPM_Variant_Value_In_Index_1_REAL_2;
prgEM.stEL3446_IO_2.MDP5001_342_Input.MDP5001_342_DPM_Variant_Value_In_Value_1_REAL		:=	MDP5001_342_DPM_Variant_Value_In_Value_1_REAL_2;
prgEM.stEL3446_IO_2.MDP5001_342_Input.MDP5001_342_DPM_Variant_Value_In_Index_2_REAL		:=	MDP5001_342_DPM_Variant_Value_In_Index_2_REAL_2;
prgEM.stEL3446_IO_2.MDP5001_342_Input.MDP5001_342_DPM_Variant_Value_In_Value_2_REAL		:=	MDP5001_342_DPM_Variant_Value_In_Value_2_REAL_2;
prgEM.stEL3446_IO_2.MDP5001_342_Input.MDP5001_342_DPM_Variant_Value_In_Index_3_REAL		:=	MDP5001_342_DPM_Variant_Value_In_Index_3_REAL_2;
prgEM.stEL3446_IO_2.MDP5001_342_Input.MDP5001_342_DPM_Variant_Value_In_Value_3_REAL		:=	MDP5001_342_DPM_Variant_Value_In_Value_3_REAL_2;
prgEM.stEL3446_IO_2.MDP5001_342_Input.MDP5001_342_DPM_Variant_Value_In_Index_4_ULINT		:=	MDP5001_342_DPM_Variant_Value_In_Index_4_ULINT_2;
prgEM.stEL3446_IO_2.MDP5001_342_Input.MDP5001_342_DPM_Variant_Value_In_Value_4_ULINT		:=	MDP5001_342_DPM_Variant_Value_In_Value_4_ULINT_2;
       
MDP5001_342_DPM_Variant_Value_Out_Index_1_REAL_2	:= 		prgEM.stEL3446_IO_2.MDP5001_342_Output.MDP5001_342_DPM_Variant_Value_Out_Index_1_REAL	;
MDP5001_342_DPM_Variant_Value_Out_Index_2_REAL_2	:= 		prgEM.stEL3446_IO_2.MDP5001_342_Output.MDP5001_342_DPM_Variant_Value_Out_Index_2_REAL	;	
MDP5001_342_DPM_Variant_Value_Out_Index_3_REAL_2	:= 		prgEM.stEL3446_IO_2.MDP5001_342_Output.MDP5001_342_DPM_Variant_Value_Out_Index_3_REAL	;
MDP5001_342_DPM_Variant_Value_Out_Index_4_ULINT_2	:= 		prgEM.stEL3446_IO_2.MDP5001_342_Output.MDP5001_342_DPM_Variant_Value_Out_Index_4_ULINT	;
MDP5001_342_DPM_Data_Data_1_2						:= 		prgEM.stEL3446_IO_2.MDP5001_342_Output.MDP5001_342_DPM_Data_Data_1	;
MDP5001_342_DPM_Data_Data_2_2						:= 		prgEM.stEL3446_IO_2.MDP5001_342_Output.MDP5001_342_DPM_Data_Data_2	;
MDP5001_342_DPM_Data_Data_3_2						:= 		prgEM.stEL3446_IO_2.MDP5001_342_Output.MDP5001_342_DPM_Data_Data_3	;
MDP5001_342_DPM_Data_Data_4_2						:= 		prgEM.stEL3446_IO_2.MDP5001_342_Output.MDP5001_342_DPM_Data_Data_4	;
MDP5001_342_DPM_Data_Data_5_2						:= 		prgEM.stEL3446_IO_2.MDP5001_342_Output.MDP5001_342_DPM_Data_Data_5	;
MDP5001_342_DPM_Data_Data_6_2						:= 		prgEM.stEL3446_IO_2.MDP5001_342_Output.MDP5001_342_DPM_Data_Data_6	;
MDP5001_342_DPM_Data_Data_7_2						:= 		prgEM.stEL3446_IO_2.MDP5001_342_Output.MDP5001_342_DPM_Data_Data_7	;
MDP5001_342_DPM_Data_Data_8_2						:= 		prgEM.stEL3446_IO_2.MDP5001_342_Output.MDP5001_342_DPM_Data_Data_8	;
MDP5001_342_DPM_Data_Data_9_2						:= 		prgEM.stEL3446_IO_2.MDP5001_342_Output.MDP5001_342_DPM_Data_Data_9	;
MDP5001_342_DPM_Data_Data_10_2						:= 		prgEM.stEL3446_IO_2.MDP5001_342_Output.MDP5001_342_DPM_Data_Data_10	;
MDP5001_342_DPM_Data_Data_11_2						:= 		prgEM.stEL3446_IO_2.MDP5001_342_Output.MDP5001_342_DPM_Data_Data_11	;
MDP5001_342_DPM_Data_Data_12_2						:= 		prgEM.stEL3446_IO_2.MDP5001_342_Output.MDP5001_342_DPM_Data_Data_12	;
MDP5001_342_DPM_Data_Data_13_2						:= 		prgEM.stEL3446_IO_2.MDP5001_342_Output.MDP5001_342_DPM_Data_Data_13	;
MDP5001_342_DPM_Data_Data_14_2						:= 		prgEM.stEL3446_IO_2.MDP5001_342_Output.MDP5001_342_DPM_Data_Data_14	;
MDP5001_342_DPM_Data_Data_15_2						:= 		prgEM.stEL3446_IO_2.MDP5001_342_Output.MDP5001_342_DPM_Data_Data_15	;
MDP5001_342_DPM_Data_Data_16_2						:= 		prgEM.stEL3446_IO_2.MDP5001_342_Output.MDP5001_342_DPM_Data_Data_16	;
MDP5001_342_DPM_Data_Data_17_2						:= 		prgEM.stEL3446_IO_2.MDP5001_342_Output.MDP5001_342_DPM_Data_Data_17	;
MDP5001_342_DPM_Data_Data_18_2						:= 		prgEM.stEL3446_IO_2.MDP5001_342_Output.MDP5001_342_DPM_Data_Data_18	;
MDP5001_342_DPM_Data_Data_19_2						:= 		prgEM.stEL3446_IO_2.MDP5001_342_Output.MDP5001_342_DPM_Data_Data_19	;
MDP5001_342_DPM_Data_Data_20_2						:= 		prgEM.stEL3446_IO_2.MDP5001_342_Output.MDP5001_342_DPM_Data_Data_20	;



prgEM.stEL3446_IO_3.MDP5001_342_Input.MDP5001_342_I1_Channel_Overcurrent					:=	MDP5001_342_I1_Channel_Overcurrent_3;
prgEM.stEL3446_IO_3.MDP5001_342_Input.MDP5001_342_I1_Channel_Inaccurate_Current			:=	MDP5001_342_I1_Channel_Inaccurate_Current_3;
prgEM.stEL3446_IO_3.MDP5001_342_Input.MDP5001_342_I1_Channel_Current_Guard_Warning		:=	MDP5001_342_I1_Channel_Current_Guard_Warning_3;
prgEM.stEL3446_IO_3.MDP5001_342_Input.MDP5001_342_I1_Channel_Current_Guard_Error			:=	MDP5001_342_I1_Channel_Current_Guard_Error_3;
prgEM.stEL3446_IO_3.MDP5001_342_Input.MDP5001_342_I1_Channel_Apparent_Power_Guard_Warning	:=	MDP5001_342_I1_Channel_Apparent_Power_Guard_Warning_3;
prgEM.stEL3446_IO_3.MDP5001_342_Input.MDP5001_342_I1_Channel_Apparent_Power_Guard_Error	:=	MDP5001_342_I1_Channel_Apparent_Power_Guard_Error_3;
prgEM.stEL3446_IO_3.MDP5001_342_Input.MDP5001_342_I1_Channel_Active_Power_Guard_Warning	:=	MDP5001_342_I1_Channel_Active_Power_Guard_Warning_3;
prgEM.stEL3446_IO_3.MDP5001_342_Input.MDP5001_342_I1_Channel_Active_Power_Guard_Error		:=	MDP5001_342_I1_Channel_Active_Power_Guard_Error_3;
prgEM.stEL3446_IO_3.MDP5001_342_Input.MDP5001_342_I1_Channel_Reactive_Power_Guard_Warning	:=	MDP5001_342_I1_Channel_Reactive_Power_Guard_Warning_3;
prgEM.stEL3446_IO_3.MDP5001_342_Input.MDP5001_342_I1_Channel_Reactive_Power_Guard_Error	:=	MDP5001_342_I1_Channel_Reactive_Power_Guard_Error_3;
prgEM.stEL3446_IO_3.MDP5001_342_Input.MDP5001_342_I1_Channel_DPM_Inaccurate				:=	MDP5001_342_I1_Channel_DPM_Inaccurate_3;
prgEM.stEL3446_IO_3.MDP5001_342_Input.MDP5001_342_I1_Channel_DPM_Timeout					:=	MDP5001_342_I1_Channel_DPM_Timeout_3;
prgEM.stEL3446_IO_3.MDP5001_342_Input.MDP5001_342_I1_Channel_TxPDO_Toggle					:=	MDP5001_342_I1_Channel_TxPDO_Toggle_3;
prgEM.stEL3446_IO_3.MDP5001_342_Input.MDP5001_342_I1_Channel_Current						:=	MDP5001_342_I1_Channel_Current_3;
prgEM.stEL3446_IO_3.MDP5001_342_Input.MDP5001_342_I1_Channel_Active_Power					:=	MDP5001_342_I1_Channel_Active_Power_3;
prgEM.stEL3446_IO_3.MDP5001_342_Input.MDP5001_342_I1_Channel_Apparent_Power				:=	MDP5001_342_I1_Channel_Apparent_Power_3;
prgEM.stEL3446_IO_3.MDP5001_342_Input.MDP5001_342_I1_Channel_Reactive_Power_Fundamental	:=	MDP5001_342_I1_Channel_Reactive_Power_Fundamental_3;
prgEM.stEL3446_IO_3.MDP5001_342_Input.MDP5001_342_I1_Channel_Active_Energy				:=	MDP5001_342_I1_Channel_Active_Energy_3;
prgEM.stEL3446_IO_3.MDP5001_342_Input.MDP5001_342_I2_Channel_Overcurrent					:=	MDP5001_342_I2_Channel_Overcurrent_3;
prgEM.stEL3446_IO_3.MDP5001_342_Input.MDP5001_342_I2_Channel_Inaccurate_Current			:=	MDP5001_342_I2_Channel_Inaccurate_Current_3;
prgEM.stEL3446_IO_3.MDP5001_342_Input.MDP5001_342_I2_Channel_Current_Guard_Warning		:=	MDP5001_342_I2_Channel_Current_Guard_Warning_3;
prgEM.stEL3446_IO_3.MDP5001_342_Input.MDP5001_342_I2_Channel_Current_Guard_Error			:=	MDP5001_342_I2_Channel_Current_Guard_Error_3;
prgEM.stEL3446_IO_3.MDP5001_342_Input.MDP5001_342_I2_Channel_Apparent_Power_Guard_Warning	:=	MDP5001_342_I2_Channel_Apparent_Power_Guard_Warning_3;
prgEM.stEL3446_IO_3.MDP5001_342_Input.MDP5001_342_I2_Channel_Apparent_Power_Guard_Error	:=	MDP5001_342_I2_Channel_Apparent_Power_Guard_Error_3;
prgEM.stEL3446_IO_3.MDP5001_342_Input.MDP5001_342_I2_Channel_Active_Power_Guard_Warning	:=	MDP5001_342_I2_Channel_Active_Power_Guard_Warning_3;
prgEM.stEL3446_IO_3.MDP5001_342_Input.MDP5001_342_I2_Channel_Active_Power_Guard_Error		:=	MDP5001_342_I2_Channel_Active_Power_Guard_Error_3;
prgEM.stEL3446_IO_3.MDP5001_342_Input.MDP5001_342_I2_Channel_Reactive_Power_Guard_Warning	:=	MDP5001_342_I2_Channel_Reactive_Power_Guard_Warning_3;
prgEM.stEL3446_IO_3.MDP5001_342_Input.MDP5001_342_I2_Channel_Reactive_Power_Guard_Error	:=	MDP5001_342_I2_Channel_Reactive_Power_Guard_Error_3;
prgEM.stEL3446_IO_3.MDP5001_342_Input.MDP5001_342_I2_Channel_DPM_Inaccurate				:=	MDP5001_342_I2_Channel_DPM_Inaccurate_3;
prgEM.stEL3446_IO_3.MDP5001_342_Input.MDP5001_342_I2_Channel_DPM_Timeout					:=	MDP5001_342_I2_Channel_DPM_Timeout_3;
prgEM.stEL3446_IO_3.MDP5001_342_Input.MDP5001_342_I2_Channel_TxPDO_Toggle					:=	MDP5001_342_I2_Channel_TxPDO_Toggle_3;
prgEM.stEL3446_IO_3.MDP5001_342_Input.MDP5001_342_I2_Channel_Current						:=	MDP5001_342_I2_Channel_Current_3;
prgEM.stEL3446_IO_3.MDP5001_342_Input.MDP5001_342_I2_Channel_Active_Power					:=	MDP5001_342_I2_Channel_Active_Power_3;
prgEM.stEL3446_IO_3.MDP5001_342_Input.MDP5001_342_I2_Channel_Apparent_Power				:=	MDP5001_342_I2_Channel_Apparent_Power_3;
prgEM.stEL3446_IO_3.MDP5001_342_Input.MDP5001_342_I2_Channel_Reactive_Power_Fundamental	:=	MDP5001_342_I2_Channel_Reactive_Power_Fundamental_3;
prgEM.stEL3446_IO_3.MDP5001_342_Input.MDP5001_342_I2_Channel_Active_Energy				:=	MDP5001_342_I2_Channel_Active_Energy_3;
prgEM.stEL3446_IO_3.MDP5001_342_Input.MDP5001_342_I3_Channel_Overcurrent					:=	MDP5001_342_I3_Channel_Overcurrent_3;
prgEM.stEL3446_IO_3.MDP5001_342_Input.MDP5001_342_I3_Channel_Inaccurate_Current			:=	MDP5001_342_I3_Channel_Inaccurate_Current_3;
prgEM.stEL3446_IO_3.MDP5001_342_Input.MDP5001_342_I3_Channel_Current_Guard_Warning		:=	MDP5001_342_I3_Channel_Current_Guard_Warning_3;
prgEM.stEL3446_IO_3.MDP5001_342_Input.MDP5001_342_I3_Channel_Current_Guard_Error			:=	MDP5001_342_I3_Channel_Current_Guard_Error_3;
prgEM.stEL3446_IO_3.MDP5001_342_Input.MDP5001_342_I3_Channel_Apparent_Power_Guard_Warning	:=	MDP5001_342_I3_Channel_Apparent_Power_Guard_Warning_3;
prgEM.stEL3446_IO_3.MDP5001_342_Input.MDP5001_342_I3_Channel_Apparent_Power_Guard_Error	:=	MDP5001_342_I3_Channel_Apparent_Power_Guard_Error_3;
prgEM.stEL3446_IO_3.MDP5001_342_Input.MDP5001_342_I3_Channel_Active_Power_Guard_Warning	:=	MDP5001_342_I3_Channel_Active_Power_Guard_Warning_3;
prgEM.stEL3446_IO_3.MDP5001_342_Input.MDP5001_342_I3_Channel_Active_Power_Guard_Error		:=	MDP5001_342_I3_Channel_Active_Power_Guard_Error_3;
prgEM.stEL3446_IO_3.MDP5001_342_Input.MDP5001_342_I3_Channel_Reactive_Power_Guard_Warning	:=	MDP5001_342_I3_Channel_Reactive_Power_Guard_Warning_3;
prgEM.stEL3446_IO_3.MDP5001_342_Input.MDP5001_342_I3_Channel_Reactive_Power_Guard_Error	:=	MDP5001_342_I3_Channel_Reactive_Power_Guard_Error_3;
prgEM.stEL3446_IO_3.MDP5001_342_Input.MDP5001_342_I3_Channel_DPM_Inaccurate				:=	MDP5001_342_I3_Channel_DPM_Inaccurate_3;
prgEM.stEL3446_IO_3.MDP5001_342_Input.MDP5001_342_I3_Channel_DPM_Timeout					:=	MDP5001_342_I3_Channel_DPM_Timeout_3;
prgEM.stEL3446_IO_3.MDP5001_342_Input.MDP5001_342_I3_Channel_TxPDO_Toggle					:=	MDP5001_342_I3_Channel_TxPDO_Toggle_3;
prgEM.stEL3446_IO_3.MDP5001_342_Input.MDP5001_342_I3_Channel_Current						:=	MDP5001_342_I3_Channel_Current_3;
prgEM.stEL3446_IO_3.MDP5001_342_Input.MDP5001_342_I3_Channel_Active_Power					:=	MDP5001_342_I3_Channel_Active_Power_3;
prgEM.stEL3446_IO_3.MDP5001_342_Input.MDP5001_342_I3_Channel_Apparent_Power				:=	MDP5001_342_I3_Channel_Apparent_Power_3;
prgEM.stEL3446_IO_3.MDP5001_342_Input.MDP5001_342_I3_Channel_Reactive_Power_Fundamental	:=	MDP5001_342_I3_Channel_Reactive_Power_Fundamental_3;
prgEM.stEL3446_IO_3.MDP5001_342_Input.MDP5001_342_I3_Channel_Active_Energy				:=	MDP5001_342_I3_Channel_Active_Energy_3;
prgEM.stEL3446_IO_3.MDP5001_342_Input.MDP5001_342_I4_Channel_Overcurrent					:=	MDP5001_342_I4_Channel_Overcurrent_3;
prgEM.stEL3446_IO_3.MDP5001_342_Input.MDP5001_342_I4_Channel_Inaccurate_Current			:=	MDP5001_342_I4_Channel_Inaccurate_Current_3;
prgEM.stEL3446_IO_3.MDP5001_342_Input.MDP5001_342_I4_Channel_Current_Guard_Warning		:=	MDP5001_342_I4_Channel_Current_Guard_Warning_3;
prgEM.stEL3446_IO_3.MDP5001_342_Input.MDP5001_342_I4_Channel_Current_Guard_Error			:=	MDP5001_342_I4_Channel_Current_Guard_Error_3;
prgEM.stEL3446_IO_3.MDP5001_342_Input.MDP5001_342_I4_Channel_Apparent_Power_Guard_Warning	:=	MDP5001_342_I4_Channel_Apparent_Power_Guard_Warning_3;
prgEM.stEL3446_IO_3.MDP5001_342_Input.MDP5001_342_I4_Channel_Apparent_Power_Guard_Error	:=	MDP5001_342_I4_Channel_Apparent_Power_Guard_Error_3;
prgEM.stEL3446_IO_3.MDP5001_342_Input.MDP5001_342_I4_Channel_Active_Power_Guard_Warning	:=	MDP5001_342_I4_Channel_Active_Power_Guard_Warning_3;
prgEM.stEL3446_IO_3.MDP5001_342_Input.MDP5001_342_I4_Channel_Active_Power_Guard_Error		:=	MDP5001_342_I4_Channel_Active_Power_Guard_Error_3;
prgEM.stEL3446_IO_3.MDP5001_342_Input.MDP5001_342_I4_Channel_Reactive_Power_Guard_Warning	:=	MDP5001_342_I4_Channel_Reactive_Power_Guard_Warning_3;
prgEM.stEL3446_IO_3.MDP5001_342_Input.MDP5001_342_I4_Channel_Reactive_Power_Guard_Error	:=	MDP5001_342_I4_Channel_Reactive_Power_Guard_Error_3;
prgEM.stEL3446_IO_3.MDP5001_342_Input.MDP5001_342_I4_Channel_DPM_Inaccurate				:=	MDP5001_342_I4_Channel_DPM_Inaccurate_3;
prgEM.stEL3446_IO_3.MDP5001_342_Input.MDP5001_342_I4_Channel_DPM_Timeout					:=	MDP5001_342_I4_Channel_DPM_Timeout_3;
prgEM.stEL3446_IO_3.MDP5001_342_Input.MDP5001_342_I4_Channel_TxPDO_Toggle					:=	MDP5001_342_I4_Channel_TxPDO_Toggle_3;
prgEM.stEL3446_IO_3.MDP5001_342_Input.MDP5001_342_I4_Channel_Current						:=	MDP5001_342_I4_Channel_Current_3;
prgEM.stEL3446_IO_3.MDP5001_342_Input.MDP5001_342_I4_Channel_Active_Power					:=	MDP5001_342_I4_Channel_Active_Power_3;
prgEM.stEL3446_IO_3.MDP5001_342_Input.MDP5001_342_I4_Channel_Apparent_Power				:=	MDP5001_342_I4_Channel_Apparent_Power_3;
prgEM.stEL3446_IO_3.MDP5001_342_Input.MDP5001_342_I4_Channel_Reactive_Power_Fundamental	:=	MDP5001_342_I4_Channel_Reactive_Power_Fundamental_3;
prgEM.stEL3446_IO_3.MDP5001_342_Input.MDP5001_342_I4_Channel_Active_Energy				:=	MDP5001_342_I4_Channel_Active_Energy_3;
prgEM.stEL3446_IO_3.MDP5001_342_Input.MDP5001_342_I5_Channel_Overcurrent					:=	MDP5001_342_I5_Channel_Overcurrent_3;
prgEM.stEL3446_IO_3.MDP5001_342_Input.MDP5001_342_I5_Channel_Inaccurate_Current			:=	MDP5001_342_I5_Channel_Inaccurate_Current_3;
prgEM.stEL3446_IO_3.MDP5001_342_Input.MDP5001_342_I5_Channel_Current_Guard_Warning		:=	MDP5001_342_I5_Channel_Current_Guard_Warning_3;
prgEM.stEL3446_IO_3.MDP5001_342_Input.MDP5001_342_I5_Channel_Current_Guard_Error			:=	MDP5001_342_I5_Channel_Current_Guard_Error_3;
prgEM.stEL3446_IO_3.MDP5001_342_Input.MDP5001_342_I5_Channel_Apparent_Power_Guard_Warning	:=	MDP5001_342_I5_Channel_Apparent_Power_Guard_Warning_3;
prgEM.stEL3446_IO_3.MDP5001_342_Input.MDP5001_342_I5_Channel_Apparent_Power_Guard_Error	:=	MDP5001_342_I5_Channel_Apparent_Power_Guard_Error_3;
prgEM.stEL3446_IO_3.MDP5001_342_Input.MDP5001_342_I5_Channel_Active_Power_Guard_Warning	:=	MDP5001_342_I5_Channel_Active_Power_Guard_Warning_3;
prgEM.stEL3446_IO_3.MDP5001_342_Input.MDP5001_342_I5_Channel_Active_Power_Guard_Error		:=	MDP5001_342_I5_Channel_Active_Power_Guard_Error_3;
prgEM.stEL3446_IO_3.MDP5001_342_Input.MDP5001_342_I5_Channel_Reactive_Power_Guard_Warning	:=	MDP5001_342_I5_Channel_Reactive_Power_Guard_Warning_3;
prgEM.stEL3446_IO_3.MDP5001_342_Input.MDP5001_342_I5_Channel_Reactive_Power_Guard_Error	:=	MDP5001_342_I5_Channel_Reactive_Power_Guard_Error_3;
prgEM.stEL3446_IO_3.MDP5001_342_Input.MDP5001_342_I5_Channel_DPM_Inaccurate				:=	MDP5001_342_I5_Channel_DPM_Inaccurate_3;
prgEM.stEL3446_IO_3.MDP5001_342_Input.MDP5001_342_I5_Channel_DPM_Timeout					:=	MDP5001_342_I5_Channel_DPM_Timeout_3;
prgEM.stEL3446_IO_3.MDP5001_342_Input.MDP5001_342_I5_Channel_TxPDO_Toggle					:=	MDP5001_342_I5_Channel_TxPDO_Toggle_3;
prgEM.stEL3446_IO_3.MDP5001_342_Input.MDP5001_342_I5_Channel_Current						:=	MDP5001_342_I5_Channel_Current_3;
prgEM.stEL3446_IO_3.MDP5001_342_Input.MDP5001_342_I5_Channel_Active_Power					:=	MDP5001_342_I5_Channel_Active_Power_3;
prgEM.stEL3446_IO_3.MDP5001_342_Input.MDP5001_342_I5_Channel_Apparent_Power				:=	MDP5001_342_I5_Channel_Apparent_Power_3;
prgEM.stEL3446_IO_3.MDP5001_342_Input.MDP5001_342_I5_Channel_Reactive_Power_Fundamental	:=	MDP5001_342_I5_Channel_Reactive_Power_Fundamental_3;
prgEM.stEL3446_IO_3.MDP5001_342_Input.MDP5001_342_I5_Channel_Active_Energy				:=	MDP5001_342_I5_Channel_Active_Energy_3;
prgEM.stEL3446_IO_3.MDP5001_342_Input.MDP5001_342_I6_Channel_Overcurrent					:=	MDP5001_342_I6_Channel_Overcurrent_3;
prgEM.stEL3446_IO_3.MDP5001_342_Input.MDP5001_342_I6_Channel_Inaccurate_Current			:=	MDP5001_342_I6_Channel_Inaccurate_Current_3;
prgEM.stEL3446_IO_3.MDP5001_342_Input.MDP5001_342_I6_Channel_Current_Guard_Warning		:=	MDP5001_342_I6_Channel_Current_Guard_Warning_3;
prgEM.stEL3446_IO_3.MDP5001_342_Input.MDP5001_342_I6_Channel_Current_Guard_Error			:=	MDP5001_342_I6_Channel_Current_Guard_Error_3;
prgEM.stEL3446_IO_3.MDP5001_342_Input.MDP5001_342_I6_Channel_Apparent_Power_Guard_Warning	:=	MDP5001_342_I6_Channel_Apparent_Power_Guard_Warning_3;
prgEM.stEL3446_IO_3.MDP5001_342_Input.MDP5001_342_I6_Channel_Apparent_Power_Guard_Error	:=	MDP5001_342_I6_Channel_Apparent_Power_Guard_Error_3;
prgEM.stEL3446_IO_3.MDP5001_342_Input.MDP5001_342_I6_Channel_Active_Power_Guard_Warning	:=	MDP5001_342_I6_Channel_Active_Power_Guard_Warning_3;
prgEM.stEL3446_IO_3.MDP5001_342_Input.MDP5001_342_I6_Channel_Active_Power_Guard_Error		:=	MDP5001_342_I6_Channel_Active_Power_Guard_Error_3;
prgEM.stEL3446_IO_3.MDP5001_342_Input.MDP5001_342_I6_Channel_Reactive_Power_Guard_Warning	:=	MDP5001_342_I6_Channel_Reactive_Power_Guard_Warning_3;
prgEM.stEL3446_IO_3.MDP5001_342_Input.MDP5001_342_I6_Channel_Reactive_Power_Guard_Error	:=	MDP5001_342_I6_Channel_Reactive_Power_Guard_Error_3;
prgEM.stEL3446_IO_3.MDP5001_342_Input.MDP5001_342_I6_Channel_DPM_Inaccurate				:=	MDP5001_342_I6_Channel_DPM_Inaccurate_3;
prgEM.stEL3446_IO_3.MDP5001_342_Input.MDP5001_342_I6_Channel_DPM_Timeout					:=	MDP5001_342_I6_Channel_DPM_Timeout_3;
prgEM.stEL3446_IO_3.MDP5001_342_Input.MDP5001_342_I6_Channel_TxPDO_Toggle					:=	MDP5001_342_I6_Channel_TxPDO_Toggle_3;
prgEM.stEL3446_IO_3.MDP5001_342_Input.MDP5001_342_I6_Channel_Current						:=	MDP5001_342_I6_Channel_Current_3;
prgEM.stEL3446_IO_3.MDP5001_342_Input.MDP5001_342_I6_Channel_Active_Power					:=	MDP5001_342_I6_Channel_Active_Power_3;
prgEM.stEL3446_IO_3.MDP5001_342_Input.MDP5001_342_I6_Channel_Apparent_Power				:=	MDP5001_342_I6_Channel_Apparent_Power_3;
prgEM.stEL3446_IO_3.MDP5001_342_Input.MDP5001_342_I6_Channel_Reactive_Power_Fundamental	:=	MDP5001_342_I6_Channel_Reactive_Power_Fundamental_3;
prgEM.stEL3446_IO_3.MDP5001_342_Input.MDP5001_342_I6_Channel_Active_Energy				:=	MDP5001_342_I6_Channel_Active_Energy_3;
prgEM.stEL3446_IO_3.MDP5001_342_Input.MDP5001_342_DPM_Variant_Value_In_TxPDO_Toggle		:=	MDP5001_342_DPM_Variant_Value_In_TxPDO_Toggle_3;
prgEM.stEL3446_IO_3.MDP5001_342_Input.MDP5001_342_DPM_Variant_Value_In_Index_1_REAL		:=	MDP5001_342_DPM_Variant_Value_In_Index_1_REAL_3;
prgEM.stEL3446_IO_3.MDP5001_342_Input.MDP5001_342_DPM_Variant_Value_In_Value_1_REAL		:=	MDP5001_342_DPM_Variant_Value_In_Value_1_REAL_3;
prgEM.stEL3446_IO_3.MDP5001_342_Input.MDP5001_342_DPM_Variant_Value_In_Index_3_REAL		:=	MDP5001_342_DPM_Variant_Value_In_Index_2_REAL_3;
prgEM.stEL3446_IO_3.MDP5001_342_Input.MDP5001_342_DPM_Variant_Value_In_Value_3_REAL		:=	MDP5001_342_DPM_Variant_Value_In_Value_2_REAL_3;
prgEM.stEL3446_IO_3.MDP5001_342_Input.MDP5001_342_DPM_Variant_Value_In_Index_3_REAL		:=	MDP5001_342_DPM_Variant_Value_In_Index_3_REAL_3;
prgEM.stEL3446_IO_3.MDP5001_342_Input.MDP5001_342_DPM_Variant_Value_In_Value_3_REAL		:=	MDP5001_342_DPM_Variant_Value_In_Value_3_REAL_3;
prgEM.stEL3446_IO_3.MDP5001_342_Input.MDP5001_342_DPM_Variant_Value_In_Index_4_ULINT		:=	MDP5001_342_DPM_Variant_Value_In_Index_4_ULINT_3;
prgEM.stEL3446_IO_3.MDP5001_342_Input.MDP5001_342_DPM_Variant_Value_In_Value_4_ULINT		:=	MDP5001_342_DPM_Variant_Value_In_Value_4_ULINT_3;

MDP5001_342_DPM_Variant_Value_Out_Index_1_REAL_3	:= 		prgEM.stEL3446_IO_3.MDP5001_342_Output.MDP5001_342_DPM_Variant_Value_Out_Index_1_REAL	;
MDP5001_342_DPM_Variant_Value_Out_Index_2_REAL_3	:= 		prgEM.stEL3446_IO_3.MDP5001_342_Output.MDP5001_342_DPM_Variant_Value_Out_Index_2_REAL	;	
MDP5001_342_DPM_Variant_Value_Out_Index_3_REAL_3	:= 		prgEM.stEL3446_IO_3.MDP5001_342_Output.MDP5001_342_DPM_Variant_Value_Out_Index_3_REAL	;
MDP5001_342_DPM_Variant_Value_Out_Index_4_ULINT_3	:= 		prgEM.stEL3446_IO_3.MDP5001_342_Output.MDP5001_342_DPM_Variant_Value_Out_Index_4_ULINT	;
MDP5001_342_DPM_Data_Data_1_3						:= 		prgEM.stEL3446_IO_3.MDP5001_342_Output.MDP5001_342_DPM_Data_Data_1	;
MDP5001_342_DPM_Data_Data_2_3						:= 		prgEM.stEL3446_IO_3.MDP5001_342_Output.MDP5001_342_DPM_Data_Data_2	;
MDP5001_342_DPM_Data_Data_3_3						:= 		prgEM.stEL3446_IO_3.MDP5001_342_Output.MDP5001_342_DPM_Data_Data_3	;
MDP5001_342_DPM_Data_Data_4_3						:= 		prgEM.stEL3446_IO_3.MDP5001_342_Output.MDP5001_342_DPM_Data_Data_4	;
MDP5001_342_DPM_Data_Data_5_3						:= 		prgEM.stEL3446_IO_3.MDP5001_342_Output.MDP5001_342_DPM_Data_Data_5	;
MDP5001_342_DPM_Data_Data_6_3						:= 		prgEM.stEL3446_IO_3.MDP5001_342_Output.MDP5001_342_DPM_Data_Data_6	;
MDP5001_342_DPM_Data_Data_7_3						:= 		prgEM.stEL3446_IO_3.MDP5001_342_Output.MDP5001_342_DPM_Data_Data_7	;
MDP5001_342_DPM_Data_Data_8_3						:= 		prgEM.stEL3446_IO_3.MDP5001_342_Output.MDP5001_342_DPM_Data_Data_8	;
MDP5001_342_DPM_Data_Data_9_3						:= 		prgEM.stEL3446_IO_3.MDP5001_342_Output.MDP5001_342_DPM_Data_Data_9	;
MDP5001_342_DPM_Data_Data_10_3						:= 		prgEM.stEL3446_IO_3.MDP5001_342_Output.MDP5001_342_DPM_Data_Data_10	;
MDP5001_342_DPM_Data_Data_11_3						:= 		prgEM.stEL3446_IO_3.MDP5001_342_Output.MDP5001_342_DPM_Data_Data_11	;
MDP5001_342_DPM_Data_Data_12_3						:= 		prgEM.stEL3446_IO_3.MDP5001_342_Output.MDP5001_342_DPM_Data_Data_12	;
MDP5001_342_DPM_Data_Data_13_3						:= 		prgEM.stEL3446_IO_3.MDP5001_342_Output.MDP5001_342_DPM_Data_Data_13	;
MDP5001_342_DPM_Data_Data_14_3						:= 		prgEM.stEL3446_IO_3.MDP5001_342_Output.MDP5001_342_DPM_Data_Data_14	;
MDP5001_342_DPM_Data_Data_15_3						:= 		prgEM.stEL3446_IO_3.MDP5001_342_Output.MDP5001_342_DPM_Data_Data_15	;
MDP5001_342_DPM_Data_Data_16_3						:= 		prgEM.stEL3446_IO_3.MDP5001_342_Output.MDP5001_342_DPM_Data_Data_16	;
MDP5001_342_DPM_Data_Data_17_3						:= 		prgEM.stEL3446_IO_3.MDP5001_342_Output.MDP5001_342_DPM_Data_Data_17	;
MDP5001_342_DPM_Data_Data_18_3						:= 		prgEM.stEL3446_IO_3.MDP5001_342_Output.MDP5001_342_DPM_Data_Data_18	;
MDP5001_342_DPM_Data_Data_19_3						:= 		prgEM.stEL3446_IO_3.MDP5001_342_Output.MDP5001_342_DPM_Data_Data_19	;
MDP5001_342_DPM_Data_Data_20_3						:= 		prgEM.stEL3446_IO_3.MDP5001_342_Output.MDP5001_342_DPM_Data_Data_20	;




prgEM.stEL3446_IO_4.MDP5001_342_Input.MDP5001_342_I1_Channel_Overcurrent					:=	MDP5001_442_I1_Channel_Overcurrent_4;
prgEM.stEL3446_IO_4.MDP5001_342_Input.MDP5001_342_I1_Channel_Inaccurate_Current			:=	MDP5001_442_I1_Channel_Inaccurate_Current_4;
prgEM.stEL3446_IO_4.MDP5001_342_Input.MDP5001_342_I1_Channel_Current_Guard_Warning		:=	MDP5001_442_I1_Channel_Current_Guard_Warning_4;
prgEM.stEL3446_IO_4.MDP5001_342_Input.MDP5001_342_I1_Channel_Current_Guard_Error			:=	MDP5001_442_I1_Channel_Current_Guard_Error_4;
prgEM.stEL3446_IO_4.MDP5001_342_Input.MDP5001_342_I1_Channel_Apparent_Power_Guard_Warning	:=	MDP5001_442_I1_Channel_Apparent_Power_Guard_Warning_4;
prgEM.stEL3446_IO_4.MDP5001_342_Input.MDP5001_342_I1_Channel_Apparent_Power_Guard_Error	:=	MDP5001_442_I1_Channel_Apparent_Power_Guard_Error_4;
prgEM.stEL3446_IO_4.MDP5001_342_Input.MDP5001_342_I1_Channel_Active_Power_Guard_Warning	:=	MDP5001_442_I1_Channel_Active_Power_Guard_Warning_4;
prgEM.stEL3446_IO_4.MDP5001_342_Input.MDP5001_342_I1_Channel_Active_Power_Guard_Error		:=	MDP5001_442_I1_Channel_Active_Power_Guard_Error_4;
prgEM.stEL3446_IO_4.MDP5001_342_Input.MDP5001_342_I1_Channel_Reactive_Power_Guard_Warning	:=	MDP5001_442_I1_Channel_Reactive_Power_Guard_Warning_4;
prgEM.stEL3446_IO_4.MDP5001_342_Input.MDP5001_342_I1_Channel_Reactive_Power_Guard_Error	:=	MDP5001_442_I1_Channel_Reactive_Power_Guard_Error_4;
prgEM.stEL3446_IO_4.MDP5001_342_Input.MDP5001_342_I1_Channel_DPM_Inaccurate				:=	MDP5001_442_I1_Channel_DPM_Inaccurate_4;
prgEM.stEL3446_IO_4.MDP5001_342_Input.MDP5001_342_I1_Channel_DPM_Timeout					:=	MDP5001_442_I1_Channel_DPM_Timeout_4;
prgEM.stEL3446_IO_4.MDP5001_342_Input.MDP5001_342_I1_Channel_TxPDO_Toggle					:=	MDP5001_442_I1_Channel_TxPDO_Toggle_4;
prgEM.stEL3446_IO_4.MDP5001_342_Input.MDP5001_342_I1_Channel_Current						:=	MDP5001_442_I1_Channel_Current_4;
prgEM.stEL3446_IO_4.MDP5001_342_Input.MDP5001_342_I1_Channel_Active_Power					:=	MDP5001_442_I1_Channel_Active_Power_4;
prgEM.stEL3446_IO_4.MDP5001_342_Input.MDP5001_342_I1_Channel_Apparent_Power				:=	MDP5001_442_I1_Channel_Apparent_Power_4;
prgEM.stEL3446_IO_4.MDP5001_342_Input.MDP5001_342_I1_Channel_Reactive_Power_Fundamental	:=	MDP5001_442_I1_Channel_Reactive_Power_Fundamental_4;
prgEM.stEL3446_IO_4.MDP5001_342_Input.MDP5001_342_I1_Channel_Active_Energy				:=	MDP5001_442_I1_Channel_Active_Energy_4;
prgEM.stEL3446_IO_4.MDP5001_342_Input.MDP5001_342_I2_Channel_Overcurrent					:=	MDP5001_442_I2_Channel_Overcurrent_4;
prgEM.stEL3446_IO_4.MDP5001_342_Input.MDP5001_342_I2_Channel_Inaccurate_Current			:=	MDP5001_442_I2_Channel_Inaccurate_Current_4;
prgEM.stEL3446_IO_4.MDP5001_342_Input.MDP5001_342_I2_Channel_Current_Guard_Warning		:=	MDP5001_442_I2_Channel_Current_Guard_Warning_4;
prgEM.stEL3446_IO_4.MDP5001_342_Input.MDP5001_342_I2_Channel_Current_Guard_Error			:=	MDP5001_442_I2_Channel_Current_Guard_Error_4;
prgEM.stEL3446_IO_4.MDP5001_342_Input.MDP5001_342_I2_Channel_Apparent_Power_Guard_Warning	:=	MDP5001_442_I2_Channel_Apparent_Power_Guard_Warning_4;
prgEM.stEL3446_IO_4.MDP5001_342_Input.MDP5001_342_I2_Channel_Apparent_Power_Guard_Error	:=	MDP5001_442_I2_Channel_Apparent_Power_Guard_Error_4;
prgEM.stEL3446_IO_4.MDP5001_342_Input.MDP5001_342_I2_Channel_Active_Power_Guard_Warning	:=	MDP5001_442_I2_Channel_Active_Power_Guard_Warning_4;
prgEM.stEL3446_IO_4.MDP5001_342_Input.MDP5001_342_I2_Channel_Active_Power_Guard_Error		:=	MDP5001_442_I2_Channel_Active_Power_Guard_Error_4;
prgEM.stEL3446_IO_4.MDP5001_342_Input.MDP5001_342_I2_Channel_Reactive_Power_Guard_Warning	:=	MDP5001_442_I2_Channel_Reactive_Power_Guard_Warning_4;
prgEM.stEL3446_IO_4.MDP5001_342_Input.MDP5001_342_I2_Channel_Reactive_Power_Guard_Error	:=	MDP5001_442_I2_Channel_Reactive_Power_Guard_Error_4;
prgEM.stEL3446_IO_4.MDP5001_342_Input.MDP5001_342_I2_Channel_DPM_Inaccurate				:=	MDP5001_442_I2_Channel_DPM_Inaccurate_4;
prgEM.stEL3446_IO_4.MDP5001_342_Input.MDP5001_342_I2_Channel_DPM_Timeout					:=	MDP5001_442_I2_Channel_DPM_Timeout_4;
prgEM.stEL3446_IO_4.MDP5001_342_Input.MDP5001_342_I2_Channel_TxPDO_Toggle					:=	MDP5001_442_I2_Channel_TxPDO_Toggle_4;
prgEM.stEL3446_IO_4.MDP5001_342_Input.MDP5001_342_I2_Channel_Current						:=	MDP5001_442_I2_Channel_Current_4;
prgEM.stEL3446_IO_4.MDP5001_342_Input.MDP5001_342_I2_Channel_Active_Power					:=	MDP5001_442_I2_Channel_Active_Power_4;
prgEM.stEL3446_IO_4.MDP5001_342_Input.MDP5001_342_I2_Channel_Apparent_Power				:=	MDP5001_442_I2_Channel_Apparent_Power_4;
prgEM.stEL3446_IO_4.MDP5001_342_Input.MDP5001_342_I2_Channel_Reactive_Power_Fundamental	:=	MDP5001_442_I2_Channel_Reactive_Power_Fundamental_4;
prgEM.stEL3446_IO_4.MDP5001_342_Input.MDP5001_342_I2_Channel_Active_Energy				:=	MDP5001_442_I2_Channel_Active_Energy_4;
prgEM.stEL3446_IO_4.MDP5001_342_Input.MDP5001_342_I3_Channel_Overcurrent					:=	MDP5001_442_I3_Channel_Overcurrent_4;
prgEM.stEL3446_IO_4.MDP5001_342_Input.MDP5001_342_I3_Channel_Inaccurate_Current			:=	MDP5001_442_I3_Channel_Inaccurate_Current_4;
prgEM.stEL3446_IO_4.MDP5001_342_Input.MDP5001_342_I3_Channel_Current_Guard_Warning		:=	MDP5001_442_I3_Channel_Current_Guard_Warning_4;
prgEM.stEL3446_IO_4.MDP5001_342_Input.MDP5001_342_I3_Channel_Current_Guard_Error			:=	MDP5001_442_I3_Channel_Current_Guard_Error_4;
prgEM.stEL3446_IO_4.MDP5001_342_Input.MDP5001_342_I3_Channel_Apparent_Power_Guard_Warning	:=	MDP5001_442_I3_Channel_Apparent_Power_Guard_Warning_4;
prgEM.stEL3446_IO_4.MDP5001_342_Input.MDP5001_342_I3_Channel_Apparent_Power_Guard_Error	:=	MDP5001_442_I3_Channel_Apparent_Power_Guard_Error_4;
prgEM.stEL3446_IO_4.MDP5001_342_Input.MDP5001_342_I3_Channel_Active_Power_Guard_Warning	:=	MDP5001_442_I3_Channel_Active_Power_Guard_Warning_4;
prgEM.stEL3446_IO_4.MDP5001_342_Input.MDP5001_342_I3_Channel_Active_Power_Guard_Error		:=	MDP5001_442_I3_Channel_Active_Power_Guard_Error_4;
prgEM.stEL3446_IO_4.MDP5001_342_Input.MDP5001_342_I3_Channel_Reactive_Power_Guard_Warning	:=	MDP5001_442_I3_Channel_Reactive_Power_Guard_Warning_4;
prgEM.stEL3446_IO_4.MDP5001_342_Input.MDP5001_342_I3_Channel_Reactive_Power_Guard_Error	:=	MDP5001_442_I3_Channel_Reactive_Power_Guard_Error_4;
prgEM.stEL3446_IO_4.MDP5001_342_Input.MDP5001_342_I3_Channel_DPM_Inaccurate				:=	MDP5001_442_I3_Channel_DPM_Inaccurate_4;
prgEM.stEL3446_IO_4.MDP5001_342_Input.MDP5001_342_I3_Channel_DPM_Timeout					:=	MDP5001_442_I3_Channel_DPM_Timeout_4;
prgEM.stEL3446_IO_4.MDP5001_342_Input.MDP5001_342_I3_Channel_TxPDO_Toggle					:=	MDP5001_442_I3_Channel_TxPDO_Toggle_4;
prgEM.stEL3446_IO_4.MDP5001_342_Input.MDP5001_342_I3_Channel_Current						:=	MDP5001_442_I3_Channel_Current_4;
prgEM.stEL3446_IO_4.MDP5001_342_Input.MDP5001_342_I3_Channel_Active_Power					:=	MDP5001_442_I3_Channel_Active_Power_4;
prgEM.stEL3446_IO_4.MDP5001_342_Input.MDP5001_342_I3_Channel_Apparent_Power				:=	MDP5001_442_I3_Channel_Apparent_Power_4;
prgEM.stEL3446_IO_4.MDP5001_342_Input.MDP5001_342_I3_Channel_Reactive_Power_Fundamental	:=	MDP5001_442_I3_Channel_Reactive_Power_Fundamental_4;
prgEM.stEL3446_IO_4.MDP5001_342_Input.MDP5001_342_I3_Channel_Active_Energy				:=	MDP5001_442_I3_Channel_Active_Energy_4;
prgEM.stEL3446_IO_4.MDP5001_342_Input.MDP5001_342_I4_Channel_Overcurrent					:=	MDP5001_442_I4_Channel_Overcurrent_4;
prgEM.stEL3446_IO_4.MDP5001_342_Input.MDP5001_342_I4_Channel_Inaccurate_Current			:=	MDP5001_442_I4_Channel_Inaccurate_Current_4;
prgEM.stEL3446_IO_4.MDP5001_342_Input.MDP5001_342_I4_Channel_Current_Guard_Warning		:=	MDP5001_442_I4_Channel_Current_Guard_Warning_4;
prgEM.stEL3446_IO_4.MDP5001_342_Input.MDP5001_342_I4_Channel_Current_Guard_Error			:=	MDP5001_442_I4_Channel_Current_Guard_Error_4;
prgEM.stEL3446_IO_4.MDP5001_342_Input.MDP5001_342_I4_Channel_Apparent_Power_Guard_Warning	:=	MDP5001_442_I4_Channel_Apparent_Power_Guard_Warning_4;
prgEM.stEL3446_IO_4.MDP5001_342_Input.MDP5001_342_I4_Channel_Apparent_Power_Guard_Error	:=	MDP5001_442_I4_Channel_Apparent_Power_Guard_Error_4;
prgEM.stEL3446_IO_4.MDP5001_342_Input.MDP5001_342_I4_Channel_Active_Power_Guard_Warning	:=	MDP5001_442_I4_Channel_Active_Power_Guard_Warning_4;
prgEM.stEL3446_IO_4.MDP5001_342_Input.MDP5001_342_I4_Channel_Active_Power_Guard_Error		:=	MDP5001_442_I4_Channel_Active_Power_Guard_Error_4;
prgEM.stEL3446_IO_4.MDP5001_342_Input.MDP5001_342_I4_Channel_Reactive_Power_Guard_Warning	:=	MDP5001_442_I4_Channel_Reactive_Power_Guard_Warning_4;
prgEM.stEL3446_IO_4.MDP5001_342_Input.MDP5001_342_I4_Channel_Reactive_Power_Guard_Error	:=	MDP5001_442_I4_Channel_Reactive_Power_Guard_Error_4;
prgEM.stEL3446_IO_4.MDP5001_342_Input.MDP5001_342_I4_Channel_DPM_Inaccurate				:=	MDP5001_442_I4_Channel_DPM_Inaccurate_4;
prgEM.stEL3446_IO_4.MDP5001_342_Input.MDP5001_342_I4_Channel_DPM_Timeout					:=	MDP5001_442_I4_Channel_DPM_Timeout_4;
prgEM.stEL3446_IO_4.MDP5001_342_Input.MDP5001_342_I4_Channel_TxPDO_Toggle					:=	MDP5001_442_I4_Channel_TxPDO_Toggle_4;
prgEM.stEL3446_IO_4.MDP5001_342_Input.MDP5001_342_I4_Channel_Current						:=	MDP5001_442_I4_Channel_Current_4;
prgEM.stEL3446_IO_4.MDP5001_342_Input.MDP5001_342_I4_Channel_Active_Power					:=	MDP5001_442_I4_Channel_Active_Power_4;
prgEM.stEL3446_IO_4.MDP5001_342_Input.MDP5001_342_I4_Channel_Apparent_Power				:=	MDP5001_442_I4_Channel_Apparent_Power_4;
prgEM.stEL3446_IO_4.MDP5001_342_Input.MDP5001_342_I4_Channel_Reactive_Power_Fundamental	:=	MDP5001_442_I4_Channel_Reactive_Power_Fundamental_4;
prgEM.stEL3446_IO_4.MDP5001_342_Input.MDP5001_342_I4_Channel_Active_Energy				:=	MDP5001_442_I4_Channel_Active_Energy_4;
prgEM.stEL3446_IO_4.MDP5001_342_Input.MDP5001_342_I5_Channel_Overcurrent					:=	MDP5001_442_I5_Channel_Overcurrent_4;
prgEM.stEL3446_IO_4.MDP5001_342_Input.MDP5001_342_I5_Channel_Inaccurate_Current			:=	MDP5001_442_I5_Channel_Inaccurate_Current_4;
prgEM.stEL3446_IO_4.MDP5001_342_Input.MDP5001_342_I5_Channel_Current_Guard_Warning		:=	MDP5001_442_I5_Channel_Current_Guard_Warning_4;
prgEM.stEL3446_IO_4.MDP5001_342_Input.MDP5001_342_I5_Channel_Current_Guard_Error			:=	MDP5001_442_I5_Channel_Current_Guard_Error_4;
prgEM.stEL3446_IO_4.MDP5001_342_Input.MDP5001_342_I5_Channel_Apparent_Power_Guard_Warning	:=	MDP5001_442_I5_Channel_Apparent_Power_Guard_Warning_4;
prgEM.stEL3446_IO_4.MDP5001_342_Input.MDP5001_342_I5_Channel_Apparent_Power_Guard_Error	:=	MDP5001_442_I5_Channel_Apparent_Power_Guard_Error_4;
prgEM.stEL3446_IO_4.MDP5001_342_Input.MDP5001_342_I5_Channel_Active_Power_Guard_Warning	:=	MDP5001_442_I5_Channel_Active_Power_Guard_Warning_4;
prgEM.stEL3446_IO_4.MDP5001_342_Input.MDP5001_342_I5_Channel_Active_Power_Guard_Error		:=	MDP5001_442_I5_Channel_Active_Power_Guard_Error_4;
prgEM.stEL3446_IO_4.MDP5001_342_Input.MDP5001_342_I5_Channel_Reactive_Power_Guard_Warning	:=	MDP5001_442_I5_Channel_Reactive_Power_Guard_Warning_4;
prgEM.stEL3446_IO_4.MDP5001_342_Input.MDP5001_342_I5_Channel_Reactive_Power_Guard_Error	:=	MDP5001_442_I5_Channel_Reactive_Power_Guard_Error_4;
prgEM.stEL3446_IO_4.MDP5001_342_Input.MDP5001_342_I5_Channel_DPM_Inaccurate				:=	MDP5001_442_I5_Channel_DPM_Inaccurate_4;
prgEM.stEL3446_IO_4.MDP5001_342_Input.MDP5001_342_I5_Channel_DPM_Timeout					:=	MDP5001_442_I5_Channel_DPM_Timeout_4;
prgEM.stEL3446_IO_4.MDP5001_342_Input.MDP5001_342_I5_Channel_TxPDO_Toggle					:=	MDP5001_442_I5_Channel_TxPDO_Toggle_4;
prgEM.stEL3446_IO_4.MDP5001_342_Input.MDP5001_342_I5_Channel_Current						:=	MDP5001_442_I5_Channel_Current_4;
prgEM.stEL3446_IO_4.MDP5001_342_Input.MDP5001_342_I5_Channel_Active_Power					:=	MDP5001_442_I5_Channel_Active_Power_4;
prgEM.stEL3446_IO_4.MDP5001_342_Input.MDP5001_342_I5_Channel_Apparent_Power				:=	MDP5001_442_I5_Channel_Apparent_Power_4;
prgEM.stEL3446_IO_4.MDP5001_342_Input.MDP5001_342_I5_Channel_Reactive_Power_Fundamental	:=	MDP5001_442_I5_Channel_Reactive_Power_Fundamental_4;
prgEM.stEL3446_IO_4.MDP5001_342_Input.MDP5001_342_I5_Channel_Active_Energy				:=	MDP5001_442_I5_Channel_Active_Energy_4;
prgEM.stEL3446_IO_4.MDP5001_342_Input.MDP5001_342_I6_Channel_Overcurrent					:=	MDP5001_442_I6_Channel_Overcurrent_4;
prgEM.stEL3446_IO_4.MDP5001_342_Input.MDP5001_342_I6_Channel_Inaccurate_Current			:=	MDP5001_442_I6_Channel_Inaccurate_Current_4;
prgEM.stEL3446_IO_4.MDP5001_342_Input.MDP5001_342_I6_Channel_Current_Guard_Warning		:=	MDP5001_442_I6_Channel_Current_Guard_Warning_4;
prgEM.stEL3446_IO_4.MDP5001_342_Input.MDP5001_342_I6_Channel_Current_Guard_Error			:=	MDP5001_442_I6_Channel_Current_Guard_Error_4;
prgEM.stEL3446_IO_4.MDP5001_342_Input.MDP5001_342_I6_Channel_Apparent_Power_Guard_Warning	:=	MDP5001_442_I6_Channel_Apparent_Power_Guard_Warning_4;
prgEM.stEL3446_IO_4.MDP5001_342_Input.MDP5001_342_I6_Channel_Apparent_Power_Guard_Error	:=	MDP5001_442_I6_Channel_Apparent_Power_Guard_Error_4;
prgEM.stEL3446_IO_4.MDP5001_342_Input.MDP5001_342_I6_Channel_Active_Power_Guard_Warning	:=	MDP5001_442_I6_Channel_Active_Power_Guard_Warning_4;
prgEM.stEL3446_IO_4.MDP5001_342_Input.MDP5001_342_I6_Channel_Active_Power_Guard_Error		:=	MDP5001_442_I6_Channel_Active_Power_Guard_Error_4;
prgEM.stEL3446_IO_4.MDP5001_342_Input.MDP5001_342_I6_Channel_Reactive_Power_Guard_Warning	:=	MDP5001_442_I6_Channel_Reactive_Power_Guard_Warning_4;
prgEM.stEL3446_IO_4.MDP5001_342_Input.MDP5001_342_I6_Channel_Reactive_Power_Guard_Error	:=	MDP5001_442_I6_Channel_Reactive_Power_Guard_Error_4;
prgEM.stEL3446_IO_4.MDP5001_342_Input.MDP5001_342_I6_Channel_DPM_Inaccurate				:=	MDP5001_442_I6_Channel_DPM_Inaccurate_4;
prgEM.stEL3446_IO_4.MDP5001_342_Input.MDP5001_342_I6_Channel_DPM_Timeout					:=	MDP5001_442_I6_Channel_DPM_Timeout_4;
prgEM.stEL3446_IO_4.MDP5001_342_Input.MDP5001_342_I6_Channel_TxPDO_Toggle					:=	MDP5001_442_I6_Channel_TxPDO_Toggle_4;
prgEM.stEL3446_IO_4.MDP5001_342_Input.MDP5001_342_I6_Channel_Current						:=	MDP5001_442_I6_Channel_Current_4;
prgEM.stEL3446_IO_4.MDP5001_342_Input.MDP5001_342_I6_Channel_Active_Power					:=	MDP5001_442_I6_Channel_Active_Power_4;
prgEM.stEL3446_IO_4.MDP5001_342_Input.MDP5001_342_I6_Channel_Apparent_Power				:=	MDP5001_442_I6_Channel_Apparent_Power_4;
prgEM.stEL3446_IO_4.MDP5001_342_Input.MDP5001_342_I6_Channel_Reactive_Power_Fundamental	:=	MDP5001_442_I6_Channel_Reactive_Power_Fundamental_4;
prgEM.stEL3446_IO_4.MDP5001_342_Input.MDP5001_342_I6_Channel_Active_Energy				:=	MDP5001_442_I6_Channel_Active_Energy_4;
prgEM.stEL3446_IO_4.MDP5001_342_Input.MDP5001_342_DPM_Variant_Value_In_TxPDO_Toggle		:=	MDP5001_442_DPM_Variant_Value_In_TxPDO_Toggle_4;
prgEM.stEL3446_IO_4.MDP5001_342_Input.MDP5001_342_DPM_Variant_Value_In_Index_1_REAL		:=	MDP5001_442_DPM_Variant_Value_In_Index_1_REAL_4;
prgEM.stEL3446_IO_4.MDP5001_342_Input.MDP5001_342_DPM_Variant_Value_In_Value_1_REAL		:=	MDP5001_442_DPM_Variant_Value_In_Value_1_REAL_4;
prgEM.stEL3446_IO_4.MDP5001_342_Input.MDP5001_342_DPM_Variant_Value_In_Index_2_REAL		:=	MDP5001_442_DPM_Variant_Value_In_Index_2_REAL_4;
prgEM.stEL3446_IO_4.MDP5001_342_Input.MDP5001_342_DPM_Variant_Value_In_Value_2_REAL		:=	MDP5001_442_DPM_Variant_Value_In_Value_2_REAL_4;
prgEM.stEL3446_IO_4.MDP5001_342_Input.MDP5001_342_DPM_Variant_Value_In_Index_3_REAL		:=	MDP5001_442_DPM_Variant_Value_In_Index_3_REAL_4;
prgEM.stEL3446_IO_4.MDP5001_342_Input.MDP5001_342_DPM_Variant_Value_In_Value_3_REAL		:=	MDP5001_442_DPM_Variant_Value_In_Value_3_REAL_4;
prgEM.stEL3446_IO_4.MDP5001_342_Input.MDP5001_342_DPM_Variant_Value_In_Index_4_ULINT		:=	MDP5001_442_DPM_Variant_Value_In_Index_4_ULINT_4;
prgEM.stEL3446_IO_4.MDP5001_342_Input.MDP5001_342_DPM_Variant_Value_In_Value_4_ULINT		:=	MDP5001_442_DPM_Variant_Value_In_Value_4_ULINT_4;

MDP5001_342_DPM_Variant_Value_Out_Index_1_REAL_4	:= 		prgEM.stEL3446_IO_4.MDP5001_342_Output.MDP5001_342_DPM_Variant_Value_Out_Index_1_REAL	;
MDP5001_342_DPM_Variant_Value_Out_Index_2_REAL_4	:= 		prgEM.stEL3446_IO_4.MDP5001_342_Output.MDP5001_342_DPM_Variant_Value_Out_Index_2_REAL	;	
MDP5001_342_DPM_Variant_Value_Out_Index_3_REAL_4	:= 		prgEM.stEL3446_IO_4.MDP5001_342_Output.MDP5001_342_DPM_Variant_Value_Out_Index_3_REAL	;
MDP5001_342_DPM_Variant_Value_Out_Index_4_ULINT_4	:= 		prgEM.stEL3446_IO_4.MDP5001_342_Output.MDP5001_342_DPM_Variant_Value_Out_Index_4_ULINT	;
MDP5001_342_DPM_Data_Data_1_4						:= 		prgEM.stEL3446_IO_4.MDP5001_342_Output.MDP5001_342_DPM_Data_Data_1	;
MDP5001_342_DPM_Data_Data_2_4						:= 		prgEM.stEL3446_IO_4.MDP5001_342_Output.MDP5001_342_DPM_Data_Data_2	;
MDP5001_342_DPM_Data_Data_3_4						:= 		prgEM.stEL3446_IO_4.MDP5001_342_Output.MDP5001_342_DPM_Data_Data_3	;
MDP5001_342_DPM_Data_Data_4_4						:= 		prgEM.stEL3446_IO_4.MDP5001_342_Output.MDP5001_342_DPM_Data_Data_4	;
MDP5001_342_DPM_Data_Data_5_4						:= 		prgEM.stEL3446_IO_4.MDP5001_342_Output.MDP5001_342_DPM_Data_Data_5	;
MDP5001_342_DPM_Data_Data_6_4						:= 		prgEM.stEL3446_IO_4.MDP5001_342_Output.MDP5001_342_DPM_Data_Data_6	;
MDP5001_342_DPM_Data_Data_7_4						:= 		prgEM.stEL3446_IO_4.MDP5001_342_Output.MDP5001_342_DPM_Data_Data_7	;
MDP5001_342_DPM_Data_Data_8_4						:= 		prgEM.stEL3446_IO_4.MDP5001_342_Output.MDP5001_342_DPM_Data_Data_8	;
MDP5001_342_DPM_Data_Data_9_4						:= 		prgEM.stEL3446_IO_4.MDP5001_342_Output.MDP5001_342_DPM_Data_Data_9	;
MDP5001_342_DPM_Data_Data_10_4						:= 		prgEM.stEL3446_IO_4.MDP5001_342_Output.MDP5001_342_DPM_Data_Data_10	;
MDP5001_342_DPM_Data_Data_11_4						:= 		prgEM.stEL3446_IO_4.MDP5001_342_Output.MDP5001_342_DPM_Data_Data_11	;
MDP5001_342_DPM_Data_Data_12_4						:= 		prgEM.stEL3446_IO_4.MDP5001_342_Output.MDP5001_342_DPM_Data_Data_12	;
MDP5001_342_DPM_Data_Data_13_4						:= 		prgEM.stEL3446_IO_4.MDP5001_342_Output.MDP5001_342_DPM_Data_Data_13	;
MDP5001_342_DPM_Data_Data_14_4						:= 		prgEM.stEL3446_IO_4.MDP5001_342_Output.MDP5001_342_DPM_Data_Data_14	;
MDP5001_342_DPM_Data_Data_15_4						:= 		prgEM.stEL3446_IO_4.MDP5001_342_Output.MDP5001_342_DPM_Data_Data_15	;
MDP5001_342_DPM_Data_Data_16_4						:= 		prgEM.stEL3446_IO_4.MDP5001_342_Output.MDP5001_342_DPM_Data_Data_16	;
MDP5001_342_DPM_Data_Data_17_4						:= 		prgEM.stEL3446_IO_4.MDP5001_342_Output.MDP5001_342_DPM_Data_Data_17	;
MDP5001_342_DPM_Data_Data_18_4						:= 		prgEM.stEL3446_IO_4.MDP5001_342_Output.MDP5001_342_DPM_Data_Data_18	;
MDP5001_342_DPM_Data_Data_19_4						:= 		prgEM.stEL3446_IO_4.MDP5001_342_Output.MDP5001_342_DPM_Data_Data_19	;
MDP5001_342_DPM_Data_Data_20_4						:= 		prgEM.stEL3446_IO_4.MDP5001_342_Output.MDP5001_342_DPM_Data_Data_20	;

END_PROGRAM

// ---- POUs/prgEM.TcPOU
PROGRAM prgEM
VAR
	fbEL3443DPM 		: FB_EM_Beckhoff_EL3443;	//EL3443 | PDO Assignment "DPM" (DPM: Distributed Power Measurement) |3-phase power measurement terminal with extended functionality
	fb_EL3446_1			: FB_EM_Beckhoff_EL3446;
	fb_EL3446_2			: FB_EM_Beckhoff_EL3446;
	fb_EL3446_3			: FB_EM_Beckhoff_EL3446;
	fb_EL3446_4			: FB_EM_Beckhoff_EL3446;
	lr_RealPower_Grid	: LREAL;						//{#lynus.ag#()}
	lr_ApparentPower_Grid: LREAL;						//{#lynus.ag#()}
	lr_ReactivePower_Grid: LREAL;						//{#lynus.ag#()}
	lr_Frequency_Grid	: LREAL;						//{#lynus.ag#()}

	lr_Voltage_L1N		: LREAL;						//{#lynus.ag#()}
	lr_Voltage_L2N		: LREAL;						//{#lynus.ag#()}
	lr_Voltage_L3N		: LREAL;						//{#lynus.ag#()}
	lr_Voltage_L1L2		: LREAL;						//{#lynus.ag#()}
	lr_Voltage_L2L3		: LREAL;						//{#lynus.ag#()}
	lr_Voltage_L3L1		: LREAL;						//{#lynus.ag#()}
 	lr_Current_L1		: LREAL;						//{#lynus.ag#()}
	lr_Current_L2		: LREAL;						//{#lynus.ag#()}
	lr_Current_L3		: LREAL;						//{#lynus.ag#()}
	lr_Power_House		: LREAL;						//{#lynus.ag#()}
	lr_RealPower_UVKeller		: LREAL;						//{#lynus.ag#()}
	lr_RealPower_UVEG			: LREAL;						//{#lynus.ag#()}
	lr_RealPower_UV1OG			: LREAL;						//{#lynus.ag#()}
	lr_RealPower_UV2OG			: LREAL;						//{#lynus.ag#()}
	lr_RealPower_Kaeltemaschine	: LREAL;						//{#lynus.ag#()}
	lr_RealPower_Spenglerei		: LREAL;						//{#lynus.ag#()}
	lr_RealPower_Werkstatt		: LREAL;						//{#lynus.ag#()}
	lr_RealPower_BueroGesamt	: LREAL;						//{#lynus.ag#()}
	
	FB_ReadMB_Zimmerei	 :FB_ModBus_100Registers_FC3_inclID;
	real_Array_Modbus_Data_Zimmerei	: ARRAY[0..49] OF REAL;


	lr_RealPower_Halle_Zimmerei		: LREAL;						//{#lynus.ag#()}
	lr_ApparentPower_Halle_Zimmerei	: LREAL;						//{#lynus.ag#()}
	lr_ReactivePower_Halle_Zimmerei	: LREAL;						//{#lynus.ag#()}
	lr_Frequency_Halle_Zimmerei		: LREAL;						//{#lynus.ag#()}
	lr_Voltage_L1N_Zimmerei			: LREAL;						//{#lynus.ag#()}
	lr_Voltage_L2N_Zimmerei			: LREAL;						//{#lynus.ag#()}
	lr_Voltage_L3N_Zimmerei			: LREAL;						//{#lynus.ag#()}
	lr_Voltage_L1L2_Zimmerei		: LREAL;						//{#lynus.ag#()}
	lr_Voltage_L2L3_Zimmerei		: LREAL;						//{#lynus.ag#()}
	lr_Voltage_L3L1_Zimmerei		: LREAL;						//{#lynus.ag#()}
 	lr_Current_L1_Zimmerei			: LREAL;						//{#lynus.ag#()}
	lr_Current_L2_Zimmerei			: LREAL;						//{#lynus.ag#()}
	lr_Current_L3_Zimmerei			: LREAL;						//{#lynus.ag#()}
	lr_RealPower_Hundegger_Zimmerei	: LREAL;						//{#lynus.ag#()}
	lr_RealPower_Spannex_Zimmerei	: LREAL;		      	     	//{#lynus.ag#()}
	lr_RealPower_Kran_Zimmerei		: LREAL;	             	   	//{#lynus.ag#()}
	lr_RealPower_Rest_Zimmerei		: LREAL;						//{#lynus.ag#()}

	FB_ReadMB_Baustoffe	 :FB_ModBus_100Registers_FC3_inclID;
	real_Array_Modbus_Data_Baustoffe	: ARRAY[0..49] OF REAL;

	lr_RealPower_Halle_Baustoffe		: LREAL;						//{#lynus.ag#()}
	lr_ApparentPower_Halle_Baustoffe	: LREAL;						//{#lynus.ag#()}
	lr_ReactivePower_Halle_Baustoffe	: LREAL;						//{#lynus.ag#()}
	lr_Frequency_Halle_Baustoffe		: LREAL;						//{#lynus.ag#()}
	lr_Voltage_L1N_Baustoffe			: LREAL;						//{#lynus.ag#()}
	lr_Voltage_L2N_Baustoffe			: LREAL;						//{#lynus.ag#()}
	lr_Voltage_L3N_Baustoffe			: LREAL;						//{#lynus.ag#()}
	lr_Voltage_L1L2_Baustoffe		: LREAL;						//{#lynus.ag#()}
	lr_Voltage_L2L3_Baustoffe		: LREAL;						//{#lynus.ag#()}
	lr_Voltage_L3L1_Baustoffe		: LREAL;						//{#lynus.ag#()}
 	lr_Current_L1_Baustoffe			: LREAL;						//{#lynus.ag#()}
	lr_Current_L2_Baustoffe			: LREAL;						//{#lynus.ag#()}
	lr_Current_L3_Baustoffe			: LREAL;						//{#lynus.ag#()}
	lr_RealPower_Kran_Baustoffe		: LREAL;	             	   	//{#lynus.ag#()}
	lr_RealPower_Rest_Baustoffe		: LREAL;						//{#lynus.ag#()}
END_VAR
VAR_INPUT
	stEL3443_IO 						: MDP5001_341_7CD731EE;
	stEL3446_IO_1 						: MDP5001_342_066CA8C6; 
	stEL3446_IO_2 						: MDP5001_342_066CA8C6; 
	stEL3446_IO_3 						: MDP5001_342_066CA8C6; 
	stEL3446_IO_4 						: MDP5001_342_066CA8C6; 
END_VAR
VAR PERSISTENT
	lr_EnergyCounter_Grid	: LREAL;						//{#lynus.ag#()}
END_VAR

// grid measurement
fbEL3443DPM(
	bEnable 	:= TRUE, 
	bInvers_CH1 := FALSE, 
	bInvers_CH2	:= FALSE, 
	bInvers_CH3	:= FALSE, 
	uiCurrentTransformerRatio:= 600,		// two cables,300:1 CTs only over one cable 
	nSlaveAddr 	:= 1001,
	b_SubIndex	:= 2,
	stEL3443_IO := ,
	pDpmData=> , 
	stDataEMPower=> , 
	stDataEMCounter=> , 
	stDataEMPowerRealTime=> , 
	stDataEMCounterRealTime=> );
fbEL3443DPM.stEL3443_IO.MDP5001_341_Input := stEL3443_IO.MDP5001_341_Input;
stEL3443_IO.MDP5001_341_Output	:= fbEL3443DPM.stEL3443_IO.MDP5001_341_Output;
 	
lr_RealPower_Grid 		:= fbEL3443DPM.stDataEMPower.lrPowerTotal; 	
lr_ApparentPower_Grid 	:= fbEL3443DPM.stDataEMPower.lrApparentPowerTotal;
lr_ReactivePower_Grid	:= fbEL3443DPM.stDataEMPower.lrReactivePowerTotal;
lr_Frequency_Grid		:= fbEL3443DPM.stDataEMPower.lrFrequency;
lr_Voltage_L1N			:= fbEL3443DPM.stDataEMPower.lrVoltageL1N;
lr_Voltage_L2N			:= fbEL3443DPM.stDataEMPower.lrVoltageL2N;
lr_Voltage_L3N			:= fbEL3443DPM.stDataEMPower.lrVoltageL3N;
lr_Voltage_L1L2			:= fbEL3443DPM.stDataEMPower.lrVoltageL1L2;
lr_Voltage_L2L3			:= fbEL3443DPM.stDataEMPower.lrVoltageL2L3;
lr_Voltage_L3L1			:= fbEL3443DPM.stDataEMPower.lrVoltageL3L1;
lr_EnergyCounter_Grid	:= fbEL3443DPM.stDataEMCounter.lrTotalCounterEnergy_Consumption;
lr_Current_L1			:= fbEL3443DPM.stDataEMPower.lrCurrentL1;
lr_Current_L2			:= fbEL3443DPM.stDataEMPower.lrCurrentL2;
lr_Current_L3			:= fbEL3443DPM.stDataEMPower.lrCurrentL3;
	 
fb_EL3446_1(
	bEnable:= TRUE , 
	bEnableVariantValues:= TRUE, 
	pDpmData:= fbEL3443DPM.pDpmData, 
	nSlaveAddr:= 1002, 
	b_SubIndex	:= 2,
	bInvers_CH1:= TRUE, 
	bInvers_CH2:= TRUE, 
	bInvers_CH3:= TRUE, 
	bInvers_CH4:= TRUE, 
	bInvers_CH5:= TRUE, 
	bInvers_CH6:= TRUE, 
	uiCurrentTransformerRatio_CH1:= 300, 
	uiCurrentTransformerRatio_CH2:= 300, 
	uiCurrentTransformerRatio_CH3:= 300, 
	uiCurrentTransformerRatio_CH4:= 300, 
	uiCurrentTransformerRatio_CH5:= 300, 
	uiCurrentTransformerRatio_CH6:= 300, 
	uiVoltagePhaseSelector_CH1:= 2, 			// phase order not 1/2/3 because voltage channel missmatch 
	uiVoltagePhaseSelector_CH2:= 3, 			// therefore signle phase channels got used
	uiVoltagePhaseSelector_CH3:= 1, 
	uiVoltagePhaseSelector_CH4:= 2, 
	uiVoltagePhaseSelector_CH5:= 3, 
	uiVoltagePhaseSelector_CH6:= 1, 
	bEnable3PhaseCH13:= FALSE, 
	bEnable3PhaseCH46:= FALSE, 
	stDataEMPowerRealTime:= fbEL3443DPM.stDataEMPowerRealTime, 
	stEL3446_IO := ,
	stDataEMPower_CH1=> , 
	stDataEMCounter_CH1=> , 
	stDataEMPowerRealTime_CH1=> , 
	stDataEMCounterRealTime_CH1=> , 
	stDataEMPower_CH2=> , 
	stDataEMCounter_CH2=> , 
	stDataEMPowerRealTime_CH2=> , 
	stDataEMCounterRealTime_CH2=> , 
	stDataEMPower_CH3=> , 
	stDataEMCounter_CH3=> , 
	stDataEMPowerRealTime_CH3=> , 
	stDataEMCounterRealTime_CH3=> , 
	stDataEMPower_CH4=> , 
	stDataEMCounter_CH4=> , 
	stDataEMPowerRealTime_CH4=> , 
	stDataEMCounterRealTime_CH4=> , 
	stDataEMPower_CH5=> , 
	stDataEMCounter_CH5=> , 
	stDataEMPowerRealTime_CH5=> , 
	stDataEMCounterRealTime_CH5=> , 
	stDataEMPower_CH6=> , 
	stDataEMCounter_CH6=> , 
	stDataEMPowerRealTime_CH6=> , 
	stDataEMCounterRealTime_CH6=> );
fb_EL3446_1.stEL3446_IO.MDP5001_342_Input := stEL3446_IO_1.MDP5001_342_Input;
stEL3446_IO_1.MDP5001_342_Output := 	fb_EL3446_1.stEL3446_IO.MDP5001_342_Output;
lr_RealPower_UVKeller	:= 	fb_EL3446_1.stDataEMPower_CH1.lrPowerConsumption + 
							fb_EL3446_1.stDataEMPower_CH2.lrPowerConsumption + 
							fb_EL3446_1.stDataEMPower_CH3.lrPowerConsumption;
lr_RealPower_UVEG		:= 	fb_EL3446_1.stDataEMPower_CH4.lrPowerConsumption + 
							fb_EL3446_1.stDataEMPower_CH5.lrPowerConsumption + 
							fb_EL3446_1.stDataEMPower_CH6.lrPowerConsumption;

fb_EL3446_2(
	bEnable:= TRUE , 
	bEnableVariantValues:= TRUE, 
	pDpmData:= fbEL3443DPM.pDpmData, 
	nSlaveAddr:= 1003, 
	b_SubIndex	:= 2,
	bInvers_CH1:= TRUE, 
	bInvers_CH2:= TRUE, 
	bInvers_CH3:= TRUE, 
	bInvers_CH4:= TRUE, 
	bInvers_CH5:= TRUE, 
	bInvers_CH6:= TRUE,	
	uiCurrentTransformerRatio_CH1:= 300, 
	uiCurrentTransformerRatio_CH2:= 300, 
	uiCurrentTransformerRatio_CH3:= 300, 
	uiCurrentTransformerRatio_CH4:= 300, 
	uiCurrentTransformerRatio_CH5:= 300, 
	uiCurrentTransformerRatio_CH6:= 300, 
	uiVoltagePhaseSelector_CH1:= 2, 			// phase order not 1/2/3 because voltage channel missmatch 
	uiVoltagePhaseSelector_CH2:= 3, 			// therefore signle phase channels got used
	uiVoltagePhaseSelector_CH3:= 1, 
	uiVoltagePhaseSelector_CH4:= 2, 
	uiVoltagePhaseSelector_CH5:= 3, 
	uiVoltagePhaseSelector_CH6:= 1, 
	bEnable3PhaseCH13:= FALSE, 
	bEnable3PhaseCH46:= FALSE, 
	stDataEMPowerRealTime:= fbEL3443DPM.stDataEMPowerRealTime, 
	stEL3446_IO := ,
	stDataEMPower_CH1=> , 
	stDataEMCounter_CH1=> , 
	stDataEMPowerRealTime_CH1=> , 
	stDataEMCounterRealTime_CH1=> , 
	stDataEMPower_CH2=> , 
	stDataEMCounter_CH2=> , 
	stDataEMPowerRealTime_CH2=> , 
	stDataEMCounterRealTime_CH2=> , 
	stDataEMPower_CH3=> , 
	stDataEMCounter_CH3=> , 
	stDataEMPowerRealTime_CH3=> , 
	stDataEMCounterRealTime_CH3=> , 
	stDataEMPower_CH4=> , 
	stDataEMCounter_CH4=> , 
	stDataEMPowerRealTime_CH4=> , 
	stDataEMCounterRealTime_CH4=> , 
	stDataEMPower_CH5=> , 
	stDataEMCounter_CH5=> , 
	stDataEMPowerRealTime_CH5=> , 
	stDataEMCounterRealTime_CH5=> , 
	stDataEMPower_CH6=> , 
	stDataEMCounter_CH6=> , 
	stDataEMPowerRealTime_CH6=> , 
	stDataEMCounterRealTime_CH6=> );
fb_EL3446_2.stEL3446_IO.MDP5001_342_Input := stEL3446_IO_2.MDP5001_342_Input;
stEL3446_IO_2.MDP5001_342_Output := 	fb_EL3446_2.stEL3446_IO.MDP5001_342_Output;
lr_RealPower_UV1OG		:= 	fb_EL3446_2.stDataEMPower_CH1.lrPowerConsumption + 
							fb_EL3446_2.stDataEMPower_CH2.lrPowerConsumption + 
							fb_EL3446_2.stDataEMPower_CH3.lrPowerConsumption;
lr_RealPower_UV2OG		:= 	fb_EL3446_2.stDataEMPower_CH4.lrPowerConsumption + 
							fb_EL3446_2.stDataEMPower_CH5.lrPowerConsumption + 
							fb_EL3446_2.stDataEMPower_CH6.lrPowerConsumption;

fb_EL3446_3(
	bEnable:= TRUE , 
	bEnableVariantValues:= TRUE, 
	pDpmData:= fbEL3443DPM.pDpmData, 
	nSlaveAddr:= 1004, 
	b_SubIndex	:= 2,
	bInvers_CH1:= TRUE, 
	bInvers_CH2:= TRUE, 
	bInvers_CH3:= TRUE, 
	bInvers_CH4:= TRUE, 
	bInvers_CH5:= TRUE, 
	bInvers_CH6:= TRUE,
	uiCurrentTransformerRatio_CH1:= 300, 
	uiCurrentTransformerRatio_CH2:= 300, 
	uiCurrentTransformerRatio_CH3:= 300, 
	uiCurrentTransformerRatio_CH4:= 300, 
	uiCurrentTransformerRatio_CH5:= 300, 
	uiCurrentTransformerRatio_CH6:= 300, 
	uiVoltagePhaseSelector_CH1:= 2, 			// phase order not 1/2/3 because voltage channel missmatch 
	uiVoltagePhaseSelector_CH2:= 3, 			// therefore signle phase channels got used
	uiVoltagePhaseSelector_CH3:= 1, 
	uiVoltagePhaseSelector_CH4:= 2, 
	uiVoltagePhaseSelector_CH5:= 3, 
	uiVoltagePhaseSelector_CH6:= 1, 
	bEnable3PhaseCH13:= FALSE, 
	bEnable3PhaseCH46:= FALSE, 
	stDataEMPowerRealTime:= fbEL3443DPM.stDataEMPowerRealTime, 
	stEL3446_IO := ,
	stDataEMPower_CH1=> , 
	stDataEMCounter_CH1=> , 
	stDataEMPowerRealTime_CH1=> , 
	stDataEMCounterRealTime_CH1=> , 
	stDataEMPower_CH2=> , 
	stDataEMCounter_CH2=> , 
	stDataEMPowerRealTime_CH2=> , 
	stDataEMCounterRealTime_CH2=> , 
	stDataEMPower_CH3=> , 
	stDataEMCounter_CH3=> , 
	stDataEMPowerRealTime_CH3=> , 
	stDataEMCounterRealTime_CH3=> , 
	stDataEMPower_CH4=> , 
	stDataEMCounter_CH4=> , 
	stDataEMPowerRealTime_CH4=> , 
	stDataEMCounterRealTime_CH4=> , 
	stDataEMPower_CH5=> , 
	stDataEMCounter_CH5=> , 
	stDataEMPowerRealTime_CH5=> , 
	stDataEMCounterRealTime_CH5=> , 
	stDataEMPower_CH6=> , 
	stDataEMCounter_CH6=> , 
	stDataEMPowerRealTime_CH6=> , 
	stDataEMCounterRealTime_CH6=> );
fb_EL3446_3.stEL3446_IO.MDP5001_342_Input := stEL3446_IO_3.MDP5001_342_Input;
stEL3446_IO_3.MDP5001_342_Output := 	fb_EL3446_3.stEL3446_IO.MDP5001_342_Output;
lr_RealPower_Kaeltemaschine	:= 	fb_EL3446_3.stDataEMPower_CH1.lrPowerConsumption + 
								fb_EL3446_3.stDataEMPower_CH2.lrPowerConsumption + 
								fb_EL3446_3.stDataEMPower_CH3.lrPowerConsumption;
lr_RealPower_Spenglerei		:= 	fb_EL3446_3.stDataEMPower_CH4.lrPowerConsumption + 
								fb_EL3446_3.stDataEMPower_CH5.lrPowerConsumption + 
								fb_EL3446_3.stDataEMPower_CH6.lrPowerConsumption;


fb_EL3446_4(
	bEnable:= TRUE , 
	bEnableVariantValues:= TRUE, 
	pDpmData:= fbEL3443DPM.pDpmData, 
	nSlaveAddr:= 1005, 
	b_SubIndex	:= 2,
	bInvers_CH1:= TRUE, 
	bInvers_CH2:= TRUE, 
	bInvers_CH3:= TRUE, 
	bInvers_CH4:= TRUE, 
	bInvers_CH5:= TRUE, 
	bInvers_CH6:= TRUE,
	uiCurrentTransformerRatio_CH1:= 300, 
	uiCurrentTransformerRatio_CH2:= 300, 
	uiCurrentTransformerRatio_CH3:= 300, 
	uiCurrentTransformerRatio_CH4:= 300, 
	uiCurrentTransformerRatio_CH5:= 300, 
	uiCurrentTransformerRatio_CH6:= 300, 
	uiVoltagePhaseSelector_CH1:= 2, 			// phase order not 1/2/3 because voltage channel missmatch 
	uiVoltagePhaseSelector_CH2:= 3, 			// therefore signle phase channels got used
	uiVoltagePhaseSelector_CH3:= 1, 
	uiVoltagePhaseSelector_CH4:= 2, 
	uiVoltagePhaseSelector_CH5:= 3, 
	uiVoltagePhaseSelector_CH6:= 1, 
	bEnable3PhaseCH13:= FALSE, 
	bEnable3PhaseCH46:= FALSE,  
	stDataEMPowerRealTime:= fbEL3443DPM.stDataEMPowerRealTime, 
	stEL3446_IO := ,
	stDataEMPower_CH1=> , 
	stDataEMCounter_CH1=> , 
	stDataEMPowerRealTime_CH1=> , 
	stDataEMCounterRealTime_CH1=> , 
	stDataEMPower_CH2=> , 
	stDataEMCounter_CH2=> , 
	stDataEMPowerRealTime_CH2=> , 
	stDataEMCounterRealTime_CH2=> , 
	stDataEMPower_CH3=> , 
	stDataEMCounter_CH3=> , 
	stDataEMPowerRealTime_CH3=> , 
	stDataEMCounterRealTime_CH3=> , 
	stDataEMPower_CH4=> , 
	stDataEMCounter_CH4=> , 
	stDataEMPowerRealTime_CH4=> , 
	stDataEMCounterRealTime_CH4=> , 
	stDataEMPower_CH5=> , 
	stDataEMCounter_CH5=> , 
	stDataEMPowerRealTime_CH5=> , 
	stDataEMCounterRealTime_CH5=> , 
	stDataEMPower_CH6=> , 
	stDataEMCounter_CH6=> , 
	stDataEMPowerRealTime_CH6=> , 
	stDataEMCounterRealTime_CH6=> );
fb_EL3446_4.stEL3446_IO.MDP5001_342_Input := stEL3446_IO_4.MDP5001_342_Input;
stEL3446_IO_4.MDP5001_342_Output := 	fb_EL3446_4.stEL3446_IO.MDP5001_342_Output;
lr_RealPower_Werkstatt	:= 		fb_EL3446_4.stDataEMPower_CH1.lrPowerConsumption + 
								fb_EL3446_4.stDataEMPower_CH2.lrPowerConsumption + 
								fb_EL3446_4.stDataEMPower_CH3.lrPowerConsumption;

lr_Power_House := lr_RealPower_Grid + prgPV.lrPowerPV - prgCS.lr_Power_CS_total;
lr_RealPower_BueroGesamt := lr_RealPower_UVKeller + lr_RealPower_UVEG + lr_RealPower_UV1OG + lr_RealPower_UV2OG;

FB_ReadMB_Zimmerei(
	m_Enable:= TRUE, 
	str_IPAdress:= '192.168.1.121', 
	w_Adress:= 12288, 
	usint_Quantity:= 100 , 
	usint_ID:= 1, 
	m_PollSuccessful=> , 
	w_Array_Received=> , 
	udint_Error_ID=> );

memcpy(ADR(real_Array_Modbus_Data_Zimmerei),ADR(FB_ReadMB_Zimmerei.w_Array_Received),200);
lr_RealPower_Halle_Zimmerei			:= REAL_TO_LREAL(real_Array_Modbus_Data_Zimmerei[0]);
lr_ApparentPower_Halle_Zimmerei		:= REAL_TO_LREAL(real_Array_Modbus_Data_Zimmerei[1]);
lr_ReactivePower_Halle_Zimmerei		:= REAL_TO_LREAL(real_Array_Modbus_Data_Zimmerei[2]);
lr_Frequency_Halle_Zimmerei			:= REAL_TO_LREAL(real_Array_Modbus_Data_Zimmerei[3]);
lr_Voltage_L1N_Zimmerei				:= REAL_TO_LREAL(real_Array_Modbus_Data_Zimmerei[4]);
lr_Voltage_L2N_Zimmerei				:= REAL_TO_LREAL(real_Array_Modbus_Data_Zimmerei[5]);
lr_Voltage_L3N_Zimmerei				:= REAL_TO_LREAL(real_Array_Modbus_Data_Zimmerei[6]);
lr_Voltage_L1L2_Zimmerei			:= REAL_TO_LREAL(real_Array_Modbus_Data_Zimmerei[7]);
lr_Voltage_L2L3_Zimmerei			:= REAL_TO_LREAL(real_Array_Modbus_Data_Zimmerei[8]);
lr_Voltage_L3L1_Zimmerei			:= REAL_TO_LREAL(real_Array_Modbus_Data_Zimmerei[9]);
lr_Current_L1_Zimmerei				:= REAL_TO_LREAL(real_Array_Modbus_Data_Zimmerei[10]);
lr_Current_L2_Zimmerei				:= REAL_TO_LREAL(real_Array_Modbus_Data_Zimmerei[11]);
lr_Current_L3_Zimmerei				:= REAL_TO_LREAL(real_Array_Modbus_Data_Zimmerei[12]);
lr_RealPower_Hundegger_Zimmerei		:= REAL_TO_LREAL(real_Array_Modbus_Data_Zimmerei[13]);
lr_RealPower_Spannex_Zimmerei		:= REAL_TO_LREAL(real_Array_Modbus_Data_Zimmerei[14]);
lr_RealPower_Kran_Zimmerei			:= REAL_TO_LREAL(real_Array_Modbus_Data_Zimmerei[15]);
lr_RealPower_Rest_Zimmerei			:= LIMIT(0,lr_RealPower_Halle_Zimmerei-lr_RealPower_Hundegger_Zimmerei-lr_RealPower_Spannex_Zimmerei-lr_RealPower_Kran_Zimmerei,500);



FB_ReadMB_Baustoffe(
	m_Enable:= TRUE, 
	str_IPAdress:= '192.168.1.122', 
	w_Adress:= 12288, 
	usint_Quantity:= 100 , 
	usint_ID:= 1, 
	m_PollSuccessful=> , 
	w_Array_Received=> , 
	udint_Error_ID=> );

memcpy(ADR(real_Array_Modbus_Data_Baustoffe),ADR(FB_ReadMB_Baustoffe.w_Array_Received),200);
lr_RealPower_Halle_Baustoffe			:= REAL_TO_LREAL(real_Array_Modbus_Data_Baustoffe[0]);
lr_ApparentPower_Halle_Baustoffe		:= REAL_TO_LREAL(real_Array_Modbus_Data_Baustoffe[1]);
lr_ReactivePower_Halle_Baustoffe		:= REAL_TO_LREAL(real_Array_Modbus_Data_Baustoffe[2]);
lr_Frequency_Halle_Baustoffe			:= REAL_TO_LREAL(real_Array_Modbus_Data_Baustoffe[3]);
lr_Voltage_L1N_Baustoffe				:= REAL_TO_LREAL(real_Array_Modbus_Data_Baustoffe[4]);
lr_Voltage_L2N_Baustoffe				:= REAL_TO_LREAL(real_Array_Modbus_Data_Baustoffe[5]);
lr_Voltage_L3N_Baustoffe				:= REAL_TO_LREAL(real_Array_Modbus_Data_Baustoffe[6]);
lr_Voltage_L1L2_Baustoffe				:= REAL_TO_LREAL(real_Array_Modbus_Data_Baustoffe[7]);
lr_Voltage_L2L3_Baustoffe				:= REAL_TO_LREAL(real_Array_Modbus_Data_Baustoffe[8]);
lr_Voltage_L3L1_Baustoffe				:= REAL_TO_LREAL(real_Array_Modbus_Data_Baustoffe[9]);
lr_Current_L1_Baustoffe					:= REAL_TO_LREAL(real_Array_Modbus_Data_Baustoffe[10]);
lr_Current_L2_Baustoffe					:= REAL_TO_LREAL(real_Array_Modbus_Data_Baustoffe[11]);
lr_Current_L3_Baustoffe					:= REAL_TO_LREAL(real_Array_Modbus_Data_Baustoffe[12]);
lr_RealPower_Kran_Baustoffe				:= REAL_TO_LREAL(real_Array_Modbus_Data_Baustoffe[13]);
lr_RealPower_Rest_Baustoffe				:= LIMIT(0,lr_RealPower_Halle_Baustoffe - lr_RealPower_Kran_Baustoffe,500);

END_PROGRAM

// ---- FBs/FB_EM_Beckhoff_EL3443.TcPOU
FUNCTION_BLOCK FB_EM_Beckhoff_EL3443
VAR_INPUT
	bEnable							: BOOL;											//Enable the function
 	bInvers_CH1						: BOOL;											//Invert the Output data from Channel 1 
	bInvers_CH2						: BOOL;											//Invert the Output data from Channel 2 
	bInvers_CH3						: BOOL;											//Invert the Output data from Channel 3
	uiCurrentTransformerRatio		: UINT;											//Current Transformer Ratio  
	nSlaveAddr						: UINT;											//EtherCat Slave ID	
 	b_SubIndex						: BYTE;											//AmsNet ID Index, typically 2 or 3
	stEL3443_IO 						: MDP5001_341_7CD731EE;
END_VAR
VAR_OUTPUT
   	pDpmData 						: POINTER TO ARRAY[1..20] OF UDINT;
	stDataEMPower					: ST_ElectricMeter_Output_Power;				//Output structure with Data from Electric Meter (Power Data) 
	stDataEMCounter					: ST_ElectricMeter_Output_Counter;				//Output structure with Data from Electric Meter (Counter Data) 
	stDataEMPowerRealTime			: ST_ElectricMeter_Output_Power;				//Output structure with Data from Electric Meter (Power Data RealTime)
	stDataEMCounterRealTime			: ST_ElectricMeter_Output_Counter;				//Output structure with Data from Electric Meter (Counter Data RealTime) 
END_VAR
VAR
	fbEM							: FB_ElectricMeter;								//Electric Meter Function
	fbEnergyCounter					: FB_EnergyCounter;								//FB energy Counter, because the KL3403 has no nice logic for the Energy value
	fbEL3443DPM 					: FB_EL3443_DPM;
	
	fb_WriteCOE_EL3443	:FB_Coe_EL3443;	
	m_COE_Done: BOOL;
	uiCurrentTransformerRatio_old		: UINT;											//Current Transformer Ratio  
	f_trig_Busy: f_trig;

	
	timDissableFunctions			: TON;											//Timer to dissable the Function after Lynus_Standards.Constants_General.tTimeDissableLynusFunctions Days without connection to the Lynus Cloud
	timResetConnectionOnGVL			: TON;											//Timer to try reset the connection Flag on the GVL. (When somebody delete the Connection Function and make only a onlinechange)
	timSetCounterValues				: TON;											//Timer to set the counter values from the KL3403 Function to the EM Function
	arrPD							: ARRAY[1..7] OF FB_PersistentData_Number;		//Function to save persistent data
	byWaitInStep					: BYTE;											//Wait in Step before start to clean data on PLC
	iStateGVLData					: INT;											//State machine to handle the data on the GVL
	diCounterForGVL					: DINT;											//Counter to clean old data on GVL
	real_Multiplier_CH1: REAL;
	real_Multiplier_CH2: REAL;
	real_Multiplier_CH3: REAL;
END_VAR

//Creator : Stefan Lackner
//Company : EfficientIO
//Date : xx.09.2023
//Version : 1.0.0.0


//With this function is possible to read out all Information from a EL3446

//NOTE for diNr.....Designation => 
//_IN = Here Data come in from other Functions or go out to other functions about the GVL
//_OUT = Here Data go out to other functions about the GVL



(*-------------------------------------------------------------Service from Backend is ready and check the connection to backen for dissabel/enable Function---------------------------------------------------------------*)

//Try to reset the variable for connection on the GVL. When all is normal then the Lynus Mqtt connection function set this variable to true in the next cycle
//When we have no connection to the backend then after Lynus_Standards.Constants_General.tTimeDissableLynusFunctions days the Function is dissabled with all of his functionalities
timResetConnectionOnGVL(IN:= NOT timResetConnectionOnGVL.Q, PT:= T#1H, Q=> , ET=> );
IF timResetConnectionOnGVL.Q THEN 
	Lynus_Standards.GVL_Communicator.bStateConnectionToEnableFunctions := FALSE; 
END_IF
IF NOT Lynus_Standards.GVL_Communicator.bStateConnectionToEnableFunctions THEN 
	timDissableFunctions.IN := TRUE; 
ELSE 
	timDissableFunctions.IN := FALSE; 
END_IF  
timDissableFunctions(IN:= , PT:= Lynus_Standards.Constants_General.tTimeDissableLynusFunctions, Q=> , ET=> );

// limit inputs
uiCurrentTransformerRatio	 := LIMIT (1,uiCurrentTransformerRatio,10000);


(*----------------------------------------------------------------------------------------EL3446 Communication----------------------------------------------------------------------------------------------*)
// write CoE values for phase selector

IF 	NOT m_COE_Done OR 	uiCurrentTransformerRatio <> uiCurrentTransformerRatio_old THEN
	fb_WriteCOE_EL3443.m_start := TRUE;
	m_COE_Done := TRUE;
	 uiCurrentTransformerRatio_old := uiCurrentTransformerRatio;
END_IF
f_trig_Busy(CLK := fb_WriteCOE_EL3443.m_Busy );
IF f_trig_Busy.Q AND (fb_WriteCOE_EL3443.m_CoE_Write_done OR fb_WriteCOE_EL3443.m_Error) THEN 
	fb_WriteCOE_EL3443.m_start := FALSE;
END_IF

fb_WriteCOE_EL3443(
	m_start:= , 
	nSlaveAddr:= nSlaveAddr, 
	b_SubIndex:= b_SubIndex,
	uiCurrentTransformerRatio:= uiCurrentTransformerRatio, 
	m_Busy=> , 
	m_CoE_Write_done=> , 
	m_Error=> , 
	udint_GetAMSNetID_Error=> , 
	udint_WriteCoE_Error=> );



fbEL3443DPM(
	bEnable:= TRUE, 
	stEL3443_IO:= stEL3443_IO , 
	stStatusTotal=> , 
	stStatusPhase_L1=> , 
	stStatusPhase_L2=> , 
	stStatusPhase_L3=> , 
	stVariantValues=> , 
	pDpmData=> pDpmData, 
	bError=> );






//Invert the Output data, because it is possible that the current transformers have been mounted in different mounting positions.
IF NOT bInvers_CH1 THEN
	real_Multiplier_CH1 := 1;
ELSE
	real_Multiplier_CH1 := -1;
END_IF
IF NOT bInvers_CH2 THEN
	real_Multiplier_CH2 := 1;
ELSE
	real_Multiplier_CH2 := -1;
END_IF
IF NOT bInvers_CH3 THEN
	real_Multiplier_CH3 := 1;
ELSE
	real_Multiplier_CH3 := -1;
END_IF


//Function
fbEM(
	bEnable:= bEnable AND NOT timDissableFunctions.Q, 
	bError:= , 
	bEnableReadOutFunction:= FALSE, 
	bWriteWithDelay:= TRUE, 
	bPowerDataInvers:= FALSE,
	bReadOutDataDone:= timSetCounterValues.Q,
	iTimeReadOutInterval:= 0, 
	iErrorCode:= , 
	iWarningCode:= , 
	lrTotalCounterEnergy_Consumption:= fbEnergyCounter.lrTotalCounterEnergy_Consumption,
	lrTotalCounterEnergy_Production:= fbEnergyCounter.lrTotalCounterEnergy_Production, 
	lrCounterEnergyT1_Consumption:= fbEnergyCounter.lrCounterEnergyT1_Consumption,
	lrCounterEnergyT2_Consumption:= fbEnergyCounter.lrCounterEnergyT2_Consumption,
	lrCounterEnergyT1_Production:= fbEnergyCounter.lrCounterEnergyT1_Production, 
	lrCounterEnergyT2_Production:= fbEnergyCounter.lrCounterEnergyT2_Production, 
	lrCurrentL1:=  REAL_TO_LREAL(fbEL3443DPM.stEL3443_IO.MDP5001_341_Input.MDP5001_341_L1_Basic_Current ),
	lrVoltageL1N:= REAL_TO_LREAL(fbEL3443DPM.stEL3443_IO.MDP5001_341_Input.MDP5001_341_L1_Basic_Voltage), 
	lrVoltageL1L2:= REAL_TO_LREAL(fbEL3443DPM.stEL3443_IO.MDP5001_341_Input.MDP5001_341_L1_Basic_Voltage * 1.73), 
	lrPowerL1:= REAL_TO_LREAL(fbEL3443DPM.stEL3443_IO.MDP5001_341_Input.MDP5001_341_L1_Power_Active_Power * real_Multiplier_CH1), 
	lrCurrentL2:=  REAL_TO_LREAL(fbEL3443DPM.stEL3443_IO.MDP5001_341_Input.MDP5001_341_L2_Basic_Current),
	lrVoltageL2N:= REAL_TO_LREAL(fbEL3443DPM.stEL3443_IO.MDP5001_341_Input.MDP5001_341_L2_Basic_Voltage), 
	lrVoltageL2L3:= REAL_TO_LREAL(fbEL3443DPM.stEL3443_IO.MDP5001_341_Input.MDP5001_341_L2_Basic_Voltage * 1.73), 
	lrPowerL2:= REAL_TO_LREAL(fbEL3443DPM.stEL3443_IO.MDP5001_341_Input.MDP5001_341_L2_Power_Active_Power  * real_Multiplier_CH2),	
	lrCurrentL3:=  REAL_TO_LREAL(fbEL3443DPM.stEL3443_IO.MDP5001_341_Input.MDP5001_341_L3_Basic_Current),
	lrVoltageL3N:= REAL_TO_LREAL(fbEL3443DPM.stEL3443_IO.MDP5001_341_Input.MDP5001_341_L3_Basic_Voltage), 
	lrVoltageL3L1:= REAL_TO_LREAL(fbEL3443DPM.stEL3443_IO.MDP5001_341_Input.MDP5001_341_L3_Basic_Voltage * 1.73), 
	lrPowerL3:= REAL_TO_LREAL(fbEL3443DPM.stEL3443_IO.MDP5001_341_Input.MDP5001_341_L3_Power_Active_Power * real_Multiplier_CH3),	

	lrPowerTotal:= fbEM.lrPowerL1+fbEM.lrPowerL2+fbEM.lrPowerL3, 
	lrFrequency:= REAL_TO_LREAL(fbEL3443DPM.stEL3443_IO.MDP5001_341_Input.MDP5001_341_Total_Basic_Frequency), 
 	lrApparentPowerTotal:= REAL_TO_LREAL(fbEL3443DPM.stEL3443_IO.MDP5001_341_Input.MDP5001_341_L1_Power_Apparent_Power + fbEL3443DPM.stEL3443_IO.MDP5001_341_Input.MDP5001_341_L2_Power_Apparent_Power + fbEL3443DPM.stEL3443_IO.MDP5001_341_Input.MDP5001_341_L3_Power_Apparent_Power) ,
	lrReactivePowerTotal:= REAL_TO_LREAL(fbEL3443DPM.stEL3443_IO.MDP5001_341_Input.MDP5001_341_L1_Power_Reactive_Power + fbEL3443DPM.stEL3443_IO.MDP5001_341_Input.MDP5001_341_L2_Power_Reactive_Power + fbEL3443DPM.stEL3443_IO.MDP5001_341_Input.MDP5001_341_L3_Power_Reactive_Power) , 
	tTimDelayOutput:= T#5S, 
	stDataEMOutPower=> stDataEMPowerRealTime, 
	stDataEMOutPowerDelay=> stDataEMPower, 
	stDataEMOutCounter=> stDataEMCounterRealTime,
	stDataEMOutCounterDelay=> stDataEMCounter,
	bReadOutMeter=> );
(*----------------------------------------------------------------------------------------Energy Counter Function----------------------------------------------------------------------------------------------*)

fbEnergyCounter(
	byActiveTariff:= 1, 
	lrPowerInput:= (fbEM.lrPowerTotal) / 1000, 
	lrTotalCounterEnergy_Consumption=> , 
	lrTotalCounterEnergy_Production=> , 
	lrCounterEnergyT1_Consumption=> , 
	lrCounterEnergyT2_Consumption=> , 
	lrCounterEnergyT1_Production=> , 
	lrCounterEnergyT2_Production=> );
(*----------------------------------------------------------------------------------------Electric Meter Function----------------------------------------------------------------------------------------------*)

